LIN {X 0,Y 524.002,Z 585.207,A -85,B 0,C 180,E1 -4848.394,E2 -4848.394} C_VEL
LIN {X 0,Y 523.999,Z 585.214,A -85,B 0,C 180,E1 -4851.516,E2 -4851.516} C_VEL
LIN {X 0,Y 524.093,Z 585.196,A -85,B 0,C 180,E1 -4854.613,E2 -4854.613} C_VEL
LIN {X 0,Y 524.102,Z 585.2,A -85,B 0,C 180,E1 -4857.694,E2 -4857.694} C_VEL
LIN {X 0,Y 524.116,Z 585.194,A -85,B 0,C 180,E1 -4860.768,E2 -4860.768} C_VEL
LIN {X 0,Y 524.067,Z 585.202,A -85,B 0,C 180,E1 -4863.075,E2 -4863.075} C_VEL
LIN {X 0,Y 524.036,Z 585.205,A -85,B 0,C 180,E1 -4866.159,E2 -4866.159} C_VEL
LIN {X 0,Y 523.994,Z 585.212,A -85,B 0,C 180,E1 -4869.262,E2 -4869.262} C_VEL
LIN {X 0,Y 523.997,Z 585.216,A -85,B 0,C 180,E1 -4871.743,E2 -4871.743} C_VEL
LIN {X 0,Y 523.981,Z 585.211,A -85,B 0,C 180,E1 -4875.052,E2 -4875.052} C_VEL
LIN {X 0,Y 523.953,Z 585.22,A -85,B 0,C 180,E1 -4877.969,E2 -4877.969} C_VEL
LIN {X 0,Y 523.961,Z 585.214,A -85,B 0,C 180,E1 -4880.41,E2 -4880.41} C_VEL
LIN {X 0,Y 523.906,Z 585.219,A -85,B 0,C 180,E1 -4882.893,E2 -4882.893} C_VEL
LIN {X 0,Y 523.944,Z 585.217,A -85,B 0,C 180,E1 -4885.419,E2 -4885.419} C_VEL
LIN {X 0,Y 523.96,Z 585.222,A -85,B 0,C 180,E1 -4887.999,E2 -4887.999} C_VEL
LIN {X 0,Y 523.942,Z 585.215,A -85,B 0,C 180,E1 -4890.857,E2 -4890.857} C_VEL
LIN {X 0,Y 523.951,Z 585.218,A -85,B 0,C 180,E1 -4893.735,E2 -4893.735} C_VEL
LIN {X 0,Y 523.915,Z 585.223,A -85,B 0,C 180,E1 -4896.405,E2 -4896.405} C_VEL
LIN {X 0,Y 523.951,Z 585.213,A -85,B 0,C 180,E1 -4899.081,E2 -4899.081} C_VEL
LIN {X 0,Y 523.958,Z 585.221,A -85,B 0,C 180,E1 -4902.118,E2 -4902.118} C_VEL
LIN {X 0,Y 523.947,Z 585.214,A -85,B 0,C 180,E1 -4905.309,E2 -4905.309} C_VEL
LIN {X 0,Y 523.914,Z 585.219,A -85,B 0,C 180,E1 -4906.923,E2 -4906.923} C_VEL
LIN {X 0,Y 523.247,Z 585.302,A -85,B 0,C 180,E1 -4907.565,E2 -4907.565} C_VEL
LIN {X 0,Y 520.402,Z 585.664,A -85,B 0,C 180,E1 -4908.607,E2 -4908.607} C_VEL
LIN {X 0,Y 517.996,Z 585.969,A -85,B 0,C 180,E1 -4909.446,E2 -4909.446} C_VEL
LIN {X 0,Y 516.96,Z 586.095,A -85,B 0,C 180,E1 -4910.093,E2 -4910.093} C_VEL
LIN {X 0,Y 516.874,Z 586.103,A -85,B 0,C 180,E1 -4910.313,E2 -4910.313} C_VEL
LIN {X 0,Y 516.878,Z 586.095,A -85,B 0,C 180,E1 -4913.342,E2 -4913.342} C_VEL
LIN {X 0,Y 516.908,Z 586.095,A -85,B 0,C 180,E1 -4916.122,E2 -4916.122} C_VEL
LIN {X 0,Y 516.887,Z 586.097,A -85,B 0,C 180,E1 -4918.936,E2 -4918.936} C_VEL
LIN {X 0,Y 516.914,Z 586.09,A -85,B 0,C 180,E1 -4921.585,E2 -4921.585} C_VEL
LIN {X 0,Y 516.927,Z 586.092,A -85,B 0,C 180,E1 -4924.211,E2 -4924.211} C_VEL
LIN {X 0,Y 516.868,Z 586.104,A -85,B 0,C 180,E1 -4926.777,E2 -4926.777} C_VEL
LIN {X 0,Y 516.935,Z 586.087,A -85,B 0,C 180,E1 -4929.732,E2 -4929.732} C_VEL
LIN {X 0,Y 516.928,Z 586.095,A -85,B 0,C 180,E1 -4932.597,E2 -4932.597} C_VEL
LIN {X 0,Y 516.939,Z 586.093,A -85,B 0,C 180,E1 -4935.03,E2 -4935.03} C_VEL
LIN {X 0,Y 516.962,Z 586.085,A -85,B 0,C 180,E1 -4938.234,E2 -4938.234} C_VEL
LIN {X 0,Y 516.967,Z 586.086,A -85,B 0,C 180,E1 -4941.4,E2 -4941.4} C_VEL
LIN {X 0,Y 516.999,Z 586.08,A -85,B 0,C 180,E1 -4943.757,E2 -4943.757} C_VEL
LIN {X 0,Y 517.011,Z 586.085,A -85,B 0,C 180,E1 -4946.883,E2 -4946.883} C_VEL
LIN {X 0,Y 517.083,Z 586.069,A -85,B 0,C 180,E1 -4950,E2 -4950} C_VEL
LIN {X 0,Y 517.012,Z 586.088,A -85,B 0,C 180,E1 -4953.117,E2 -4953.117} C_VEL
LIN {X 0,Y 517,Z 586.079,A -85,B 0,C 180,E1 -4956.243,E2 -4956.243} C_VEL
LIN {X 0,Y 516.95,Z 586.093,A -85,B 0,C 180,E1 -4959.389,E2 -4959.389} C_VEL
LIN {X 0,Y 516.949,Z 586.088,A -85,B 0,C 180,E1 -4961.807,E2 -4961.807} C_VEL
LIN {X 0,Y 516.941,Z 586.093,A -85,B 0,C 180,E1 -4965.146,E2 -4965.146} C_VEL
LIN {X 0,Y 516.922,Z 586.089,A -85,B 0,C 180,E1 -4968.222,E2 -4968.222} C_VEL
LIN {X 0,Y 516.908,Z 586.093,A -85,B 0,C 180,E1 -4970.701,E2 -4970.701} C_VEL
LIN {X 0,Y 516.867,Z 586.103,A -85,B 0,C 180,E1 -4973.223,E2 -4973.223} C_VEL
LIN {X 0,Y 516.991,Z 586.242,A -85,B 0,C 180,E1 -4975.877,E2 -4975.877} C_VEL
LIN {X 0,Y 517.471,Z 590.741,A -85,B 0,C 180,E1 -4976.845,E2 -4976.845} C_VEL
LIN {X 0,Y 517.158,Z 604.413,A -85,B 0,C 180,E1 -4979.701,E2 -4979.701} C_VEL
LIN {X 0,Y 519.054,Z 615.156,A -85,B 0,C 180,E1 -4979.913,E2 -4979.913} C_VEL
LIN {X 0,Y 518.599,Z 710.584,A -85,B 0,C 180,E1 -4981.261,E2 -4981.261} C_VEL
LIN {X 0,Y 518.426,Z 723.815,A -85,B 0,C 180,E1 -4981.605,E2 -4981.605} C_VEL
LIN {X 0,Y 518.161,Z 736.677,A -85,B 0,C 180,E1 -4982.107,E2 -4982.107} C_VEL
LIN {X 0,Y 517.866,Z 748.841,A -85,B 0,C 180,E1 -4982.754,E2 -4982.754} C_VEL
LIN {X 0,Y 517.561,Z 759.435,A -85,B 0,C 180,E1 -4983.479,E2 -4983.479} C_VEL
LIN {X 0,Y 517.257,Z 770.01,A -85,B 0,C 180,E1 -4984.382,E2 -4984.382} C_VEL
LIN {X 0,Y 516.977,Z 779.197,A -85,B 0,C 180,E1 -4985.348,E2 -4985.348} C_VEL
LIN {X 0,Y 516.739,Z 787.518,A -85,B 0,C 180,E1 -4986.424,E2 -4986.424} C_VEL
LIN {X 0,Y 516.537,Z 794.357,A -85,B 0,C 180,E1 -4987.507,E2 -4987.507} C_VEL
LIN {X 0,Y 516.404,Z 800.707,A -85,B 0,C 180,E1 -4988.757,E2 -4988.757} C_VEL
LIN {X 0,Y 516.359,Z 804.811,A -85,B 0,C 180,E1 -4989.768,E2 -4989.768} C_VEL
LIN {X 0,Y 516.282,Z 808.167,A -85,B 0,C 180,E1 -4990.798,E2 -4990.798} C_VEL
LIN {X 0,Y 516.285,Z 810.728,A -85,B 0,C 180,E1 -4991.836,E2 -4991.836} C_VEL
LIN {X 0,Y 516.186,Z 812.578,A -85,B 0,C 180,E1 -4992.902,E2 -4992.902} C_VEL
LIN {X 0,Y 516.176,Z 813.697,A -85,B 0,C 180,E1 -4993.977,E2 -4993.977} C_VEL
LIN {X 0,Y 516.182,Z 814.083,A -85,B 0,C 180,E1 -4995.071,E2 -4995.071} C_VEL
LIN {X 0,Y 516.17,Z 813.652,A -85,B 0,C 180,E1 -4996.188,E2 -4996.188} C_VEL
LIN {X 0,Y 516.201,Z 812.387,A -85,B 0,C 180,E1 -4997.323,E2 -4997.323} C_VEL
LIN {X 0,Y 516.292,Z 810.232,A -85,B 0,C 180,E1 -4998.475,E2 -4998.475} C_VEL
LIN {X 0,Y 516.316,Z 807.046,A -85,B 0,C 180,E1 -4999.662,E2 -4999.662} C_VEL
LIN {X 0,Y 516.388,Z 802.692,A -85,B 0,C 180,E1 -5000.873,E2 -5000.873} C_VEL
LIN {X 0,Y 516.52,Z 796.26,A -85,B 0,C 180,E1 -5002.245,E2 -5002.245} C_VEL
LIN {X 0,Y 516.726,Z 789.583,A -85,B 0,C 180,E1 -5003.364,E2 -5003.364} C_VEL
LIN {X 0,Y 516.944,Z 781.446,A -85,B 0,C 180,E1 -5004.472,E2 -5004.472} C_VEL
LIN {X 0,Y 517.213,Z 772.092,A -85,B 0,C 180,E1 -5005.509,E2 -5005.509} C_VEL
LIN {X 0,Y 517.515,Z 762.175,A -85,B 0,C 180,E1 -5006.4,E2 -5006.4} C_VEL
LIN {X 0,Y 517.792,Z 752.322,A -85,B 0,C 180,E1 -5007.118,E2 -5007.118} C_VEL
LIN {X 0,Y 518.056,Z 739.976,A -85,B 0,C 180,E1 -5007.828,E2 -5007.828} C_VEL
LIN {X 0,Y 518.326,Z 727.745,A -85,B 0,C 180,E1 -5008.354,E2 -5008.354} C_VEL
LIN {X 0,Y 518.545,Z 714.491,A -85,B 0,C 180,E1 -5008.744,E2 -5008.744} C_VEL
LIN {X 0,Y 518.678,Z 697.737,A -85,B 0,C 180,E1 -5009.024,E2 -5009.024} C_VEL
LIN {X 0,Y 519.018,Z 614.494,A -85,B 0,C 180,E1 -5010.186,E2 -5010.186} C_VEL
LIN {X 0,Y 517.169,Z 604.571,A -85,B 0,C 180,E1 -5010.395,E2 -5010.395} C_VEL
LIN {X 0,Y 517.523,Z 590.393,A -85,B 0,C 180,E1 -5013.376,E2 -5013.376} C_VEL
LIN {X 0,Y 516.976,Z 586.092,A -85,B 0,C 180,E1 -5014.322,E2 -5014.322} C_VEL
LIN {X 0,Y 516.859,Z 586.1,A -85,B 0,C 180,E1 -5017.622,E2 -5017.622} C_VEL
LIN {X 0,Y 516.922,Z 586.094,A -85,B 0,C 180,E1 -5020.13,E2 -5020.13} C_VEL
LIN {X 0,Y 516.92,Z 586.099,A -85,B 0,C 180,E1 -5022.596,E2 -5022.596} C_VEL
LIN {X 0,Y 516.93,Z 586.094,A -85,B 0,C 180,E1 -5025.03,E2 -5025.03} C_VEL
LIN {X 0,Y 516.993,Z 586.084,A -85,B 0,C 180,E1 -5028.235,E2 -5028.235} C_VEL
LIN {X 0,Y 516.964,Z 586.087,A -85,B 0,C 180,E1 -5031.4,E2 -5031.4} C_VEL
LIN {X 0,Y 517.055,Z 586.08,A -85,B 0,C 180,E1 -5034.541,E2 -5034.541} C_VEL
LIN {X 0,Y 517.075,Z 586.071,A -85,B 0,C 180,E1 -5037.663,E2 -5037.663} C_VEL
LIN {X 0,Y 517.086,Z 586.078,A -85,B 0,C 180,E1 -5040.779,E2 -5040.779} C_VEL
LIN {X 0,Y 517.009,Z 586.084,A -85,B 0,C 180,E1 -5043.117,E2 -5043.117} C_VEL
LIN {X 0,Y 517.006,Z 586.08,A -85,B 0,C 180,E1 -5046.244,E2 -5046.244} C_VEL
LIN {X 0,Y 516.951,Z 586.089,A -85,B 0,C 180,E1 -5049.39,E2 -5049.39} C_VEL
LIN {X 0,Y 516.974,Z 586.084,A -85,B 0,C 180,E1 -5051.825,E2 -5051.825} C_VEL
LIN {X 0,Y 516.934,Z 586.095,A -85,B 0,C 180,E1 -5055.147,E2 -5055.147} C_VEL
LIN {X 0,Y 516.917,Z 586.091,A -85,B 0,C 180,E1 -5058.223,E2 -5058.223} C_VEL
LIN {X 0,Y 516.905,Z 586.095,A -85,B 0,C 180,E1 -5060.702,E2 -5060.702} C_VEL
LIN {X 0,Y 516.903,Z 586.092,A -85,B 0,C 180,E1 -5064.073,E2 -5064.073} C_VEL
LIN {X 0,Y 516.922,Z 586.09,A -85,B 0,C 180,E1 -5066.658,E2 -5066.658} C_VEL
LIN {X 0,Y 516.918,Z 586.095,A -85,B 0,C 180,E1 -5069.527,E2 -5069.527} C_VEL
LIN {X 0,Y 516.895,Z 586.091,A -85,B 0,C 180,E1 -5072.545,E2 -5072.545} C_VEL
LIN {X 0,Y 516.878,Z 586.102,A -85,B 0,C 180,E1 -5075.333,E2 -5075.333} C_VEL
LIN {X 0,Y 516.88,Z 586.096,A -85,B 0,C 180,E1 -5077.945,E2 -5077.945} C_VEL
LIN {X 0,Y 516.881,Z 586.095,A -85,B 0,C 180,E1 -5080.742,E2 -5080.742} C_VEL
LIN {X 0,Y 516.901,Z 586.094,A -85,B 0,C 180,E1 -5082.83,E2 -5082.83} C_VEL
LIN {X 0,Y 516.919,Z 586.094,A -85,B 0,C 180,E1 -5085.011,E2 -5085.011} C_VEL
LIN {X 0,Y 516.919,Z 586.091,A -85,B 0,C 180,E1 -5088.399,E2 -5088.399} C_VEL
LIN {X 0,Y 516.884,Z 586.101,A -85,B 0,C 180,E1 -5091.286,E2 -5091.286} C_VEL
LIN {X 0,Y 516.891,Z 586.096,A -85,B 0,C 180,E1 -5094.222,E2 -5094.222} C_VEL
LIN {X 0,Y 516.896,Z 586.097,A -85,B 0,C 180,E1 -5097.054,E2 -5097.054} C_VEL
LIN {X 0,Y 516.892,Z 586.101,A -85,B 0,C 180,E1 -5099.797,E2 -5099.797} C_VEL
LIN {X 0,Y 516.926,Z 586.093,A -85,B 0,C 180,E1 -5102.468,E2 -5102.468} C_VEL
LIN {X 0,Y 516.978,Z 586.172,A -85,B 0,C 180,E1 -5104.7,E2 -5104.7} C_VEL
LIN {X 0,Y 518.662,Z 595.377,A -85,B 0,C 180,E1 -5106.227,E2 -5106.227} C_VEL
LIN {X 0,Y 518.399,Z 608.933,A -85,B 0,C 180,E1 -5108.32,E2 -5108.32} C_VEL
LIN {X 0,Y 517.851,Z 630.646,A -85,B 0,C 180,E1 -5111.607,E2 -5111.607} C_VEL
LIN {X 0,Y 517.378,Z 650.872,A -85,B 0,C 180,E1 -5114.637,E2 -5114.637} C_VEL
LIN {X 0,Y 519.074,Z 662.348,A -85,B 0,C 180,E1 -5114.85,E2 -5114.85} C_VEL
LIN {X 0,Y 518.618,Z 760.232,A -85,B 0,C 180,E1 -5116.232,E2 -5116.232} C_VEL
LIN {X 0,Y 518.373,Z 773.275,A -85,B 0,C 180,E1 -5116.575,E2 -5116.575} C_VEL
LIN {X 0,Y 518.109,Z 785.905,A -85,B 0,C 180,E1 -5117.067,E2 -5117.067} C_VEL
LIN {X 0,Y 517.868,Z 798.122,A -85,B 0,C 180,E1 -5117.72,E2 -5117.72} C_VEL
LIN {X 0,Y 517.519,Z 810.11,A -85,B 0,C 180,E1 -5118.545,E2 -5118.545} C_VEL
LIN {X 0,Y 517.193,Z 820.364,A -85,B 0,C 180,E1 -5119.43,E2 -5119.43} C_VEL
LIN {X 0,Y 516.939,Z 829.589,A -85,B 0,C 180,E1 -5120.413,E2 -5120.413} C_VEL
LIN {X 0,Y 516.717,Z 838.577,A -85,B 0,C 180,E1 -5121.593,E2 -5121.593} C_VEL
LIN {X 0,Y 516.511,Z 845.809,A -85,B 0,C 180,E1 -5122.77,E2 -5122.77} C_VEL
LIN {X 0,Y 516.427,Z 850.677,A -85,B 0,C 180,E1 -5123.75,E2 -5123.75} C_VEL
LIN {X 0,Y 516.314,Z 855.373,A -85,B 0,C 180,E1 -5124.924,E2 -5124.924} C_VEL
LIN {X 0,Y 516.355,Z 858.958,A -85,B 0,C 180,E1 -5126.098,E2 -5126.098} C_VEL
LIN {X 0,Y 516.283,Z 860.807,A -85,B 0,C 180,E1 -5126.879,E2 -5126.879} C_VEL
LIN {X 0,Y 516.26,Z 862.193,A -85,B 0,C 180,E1 -5127.659,E2 -5127.659} C_VEL
LIN {X 0,Y 516.16,Z 863.785,A -85,B 0,C 180,E1 -5129.22,E2 -5129.22} C_VEL
LIN {X 0,Y 516.154,Z 864,A -85,B 0,C 180,E1 -5130,E2 -5130} C_VEL
LIN {X 0,Y 516.192,Z 863.183,A -85,B 0,C 180,E1 -5131.56,E2 -5131.56} C_VEL
LIN {X 0,Y 516.26,Z 862.195,A -85,B 0,C 180,E1 -5132.341,E2 -5132.341} C_VEL
LIN {X 0,Y 516.283,Z 860.81,A -85,B 0,C 180,E1 -5133.121,E2 -5133.121} C_VEL
LIN {X 0,Y 516.344,Z 857.895,A -85,B 0,C 180,E1 -5134.293,E2 -5134.293} C_VEL
LIN {X 0,Y 516.405,Z 853.948,A -85,B 0,C 180,E1 -5135.467,E2 -5135.467} C_VEL
LIN {X 0,Y 516.486,Z 848.017,A -85,B 0,C 180,E1 -5136.807,E2 -5136.807} C_VEL
LIN {X 0,Y 516.641,Z 841.154,A -85,B 0,C 180,E1 -5138.015,E2 -5138.015} C_VEL
LIN {X 0,Y 516.845,Z 832.837,A -85,B 0,C 180,E1 -5139.194,E2 -5139.194} C_VEL
LIN {X 0,Y 517.076,Z 824.312,A -85,B 0,C 180,E1 -5140.177,E2 -5140.177} C_VEL
LIN {X 0,Y 517.433,Z 813.782,A -85,B 0,C 180,E1 -5141.16,E2 -5141.16} C_VEL
LIN {X 0,Y 517.703,Z 802.188,A -85,B 0,C 180,E1 -5142.029,E2 -5142.029} C_VEL
LIN {X 0,Y 518.026,Z 791.939,A -85,B 0,C 180,E1 -5142.636,E2 -5142.636} C_VEL
LIN {X 0,Y 518.279,Z 780.195,A -85,B 0,C 180,E1 -5143.178,E2 -5143.178} C_VEL
LIN {X 0,Y 518.473,Z 767.577,A -85,B 0,C 180,E1 -5143.597,E2 -5143.597} C_VEL
LIN {X 0,Y 518.677,Z 754.739,A -85,B 0,C 180,E1 -5143.866,E2 -5143.866} C_VEL
LIN {X 0,Y 519.021,Z 661.489,A -85,B 0,C 180,E1 -5145.165,E2 -5145.165} C_VEL
LIN {X 0,Y 517.369,Z 650.938,A -85,B 0,C 180,E1 -5145.374,E2 -5145.374} C_VEL
LIN {X 0,Y 517.925,Z 629.521,A -85,B 0,C 180,E1 -5148.595,E2 -5148.595} C_VEL
LIN {X 0,Y 518.425,Z 609.247,A -85,B 0,C 180,E1 -5151.679,E2 -5151.679} C_VEL
LIN {X 0,Y 518.736,Z 595.718,A -85,B 0,C 180,E1 -5153.769,E2 -5153.769} C_VEL
LIN {X 0,Y 516.951,Z 586.092,A -85,B 0,C 180,E1 -5155.409,E2 -5155.409} C_VEL
LIN {X 0,Y 516.92,Z 586.099,A -85,B 0,C 180,E1 -5158.414,E2 -5158.414} C_VEL
LIN {X 0,Y 516.889,Z 586.096,A -85,B 0,C 180,E1 -5161.109,E2 -5161.109} C_VEL
LIN {X 0,Y 516.912,Z 586.093,A -85,B 0,C 180,E1 -5163.966,E2 -5163.966} C_VEL
LIN {X 0,Y 516.882,Z 586.1,A -85,B 0,C 180,E1 -5166.745,E2 -5166.745} C_VEL
LIN {X 0,Y 516.901,Z 586.092,A -85,B 0,C 180,E1 -5169.718,E2 -5169.718} C_VEL
LIN {X 0,Y 516.915,Z 586.09,A -85,B 0,C 180,E1 -5171.774,E2 -5171.774} C_VEL
LIN {X 0,Y 516.919,Z 586.094,A -85,B 0,C 180,E1 -5175.009,E2 -5175.009} C_VEL
LIN {X 0,Y 516.913,Z 586.095,A -85,B 0,C 180,E1 -5178.397,E2 -5178.397} C_VEL
LIN {X 0,Y 516.879,Z 586.097,A -85,B 0,C 180,E1 -5181.283,E2 -5181.283} C_VEL
LIN {X 0,Y 516.885,Z 586.095,A -85,B 0,C 180,E1 -5184.22,E2 -5184.22} C_VEL
LIN {X 0,Y 516.891,Z 586.099,A -85,B 0,C 180,E1 -5187.052,E2 -5187.052} C_VEL
LIN {X 0,Y 516.895,Z 586.093,A -85,B 0,C 180,E1 -5189.796,E2 -5189.796} C_VEL
LIN {X 0,Y 516.923,Z 586.092,A -85,B 0,C 180,E1 -5192.467,E2 -5192.467} C_VEL
LIN {X 0,Y 516.904,Z 586.1,A -85,B 0,C 180,E1 -5195.071,E2 -5195.071} C_VEL
LIN {X 0,Y 516.878,Z 586.096,A -85,B 0,C 180,E1 -5198.462,E2 -5198.462} C_VEL
LIN {X 0,Y 516.897,Z 586.099,A -85,B 0,C 180,E1 -5200.954,E2 -5200.954} C_VEL
LIN {X 0,Y 516.908,Z 586.096,A -85,B 0,C 180,E1 -5203.41,E2 -5203.41} C_VEL
LIN {X 0,Y 516.886,Z 586.095,A -85,B 0,C 180,E1 -5205.833,E2 -5205.833} C_VEL
LIN {X 0,Y 516.948,Z 586.092,A -85,B 0,C 180,E1 -5209.027,E2 -5209.027} C_VEL
LIN {X 0,Y 516.969,Z 586.083,A -85,B 0,C 180,E1 -5212.186,E2 -5212.186} C_VEL
LIN {X 0,Y 517.038,Z 586.075,A -85,B 0,C 180,E1 -5214.54,E2 -5214.54} C_VEL
LIN {X 0,Y 517.074,Z 586.076,A -85,B 0,C 180,E1 -5217.663,E2 -5217.663} C_VEL
LIN {X 0,Y 517.086,Z 586.07,A -85,B 0,C 180,E1 -5220.778,E2 -5220.778} C_VEL
LIN {X 0,Y 517.008,Z 586.082,A -85,B 0,C 180,E1 -5223.117,E2 -5223.117} C_VEL
LIN {X 0,Y 517,Z 586.08,A -85,B 0,C 180,E1 -5226.243,E2 -5226.243} C_VEL
LIN {X 0,Y 516.948,Z 586.092,A -85,B 0,C 180,E1 -5229.389,E2 -5229.389} C_VEL
LIN {X 0,Y 516.946,Z 586.094,A -85,B 0,C 180,E1 -5231.81,E2 -5231.81} C_VEL
LIN {X 0,Y 516.932,Z 586.09,A -85,B 0,C 180,E1 -5235.146,E2 -5235.146} C_VEL
LIN {X 0,Y 516.915,Z 586.093,A -85,B 0,C 180,E1 -5238.222,E2 -5238.222} C_VEL
LIN {X 0,Y 516.902,Z 586.092,A -85,B 0,C 180,E1 -5240.701,E2 -5240.701} C_VEL
LIN {X 0,Y 516.9,Z 586.099,A -85,B 0,C 180,E1 -5244.072,E2 -5244.072} C_VEL
LIN {X 0,Y 516.919,Z 586.09,A -85,B 0,C 180,E1 -5246.658,E2 -5246.658} C_VEL
LIN {X 0,Y 516.914,Z 586.093,A -85,B 0,C 180,E1 -5249.527,E2 -5249.527} C_VEL
LIN {X 0,Y 516.89,Z 586.096,A -85,B 0,C 180,E1 -5252.545,E2 -5252.545} C_VEL
LIN {X 0,Y 516.873,Z 586.096,A -85,B 0,C 180,E1 -5255.333,E2 -5255.333} C_VEL
LIN {X 0,Y 516.873,Z 586.102,A -85,B 0,C 180,E1 -5257.944,E2 -5257.944} C_VEL
LIN {X 0,Y 516.908,Z 586.093,A -85,B 0,C 180,E1 -5260.739,E2 -5260.739} C_VEL
LIN {X 0,Y 516.875,Z 586.099,A -85,B 0,C 180,E1 -5263.903,E2 -5263.903} C_VEL
LIN {X 0,Y 516.874,Z 586.102,A -85,B 0,C 180,E1 -5266.107,E2 -5266.107} C_VEL
LIN {X 0,Y 516.909,Z 586.099,A -85,B 0,C 180,E1 -5268.399,E2 -5268.399} C_VEL
LIN {X 0,Y 516.874,Z 586.103,A -85,B 0,C 180,E1 -5270.313,E2 -5270.313} C_VEL
LIN {X 0,Y 516.205,Z 586.182,A -85,B 0,C 180,E1 -5270.963,E2 -5270.963} C_VEL
LIN {X 0,Y 513.359,Z 586.537,A -85,B 0,C 180,E1 -5272.019,E2 -5272.019} C_VEL
LIN {X 0,Y 510.952,Z 586.836,A -85,B 0,C 180,E1 -5272.869,E2 -5272.869} C_VEL
LIN {X 0,Y 509.912,Z 586.963,A -85,B 0,C 180,E1 -5273.526,E2 -5273.526} C_VEL
LIN {X 0,Y 509.825,Z 586.974,A -85,B 0,C 180,E1 -5273.748,E2 -5273.748} C_VEL
LIN {X 0,Y 509.858,Z 586.978,A -85,B 0,C 180,E1 -5276.54,E2 -5276.54} C_VEL
LIN {X 0,Y 509.84,Z 586.972,A -85,B 0,C 180,E1 -5279.335,E2 -5279.335} C_VEL
LIN {X 0,Y 509.889,Z 586.968,A -85,B 0,C 180,E1 -5282.055,E2 -5282.055} C_VEL
LIN {X 0,Y 509.872,Z 586.976,A -85,B 0,C 180,E1 -5284.704,E2 -5284.704} C_VEL
LIN {X 0,Y 509.832,Z 586.973,A -85,B 0,C 180,E1 -5287.455,E2 -5287.455} C_VEL
LIN {X 0,Y 509.913,Z 586.962,A -85,B 0,C 180,E1 -5289.845,E2 -5289.845} C_VEL
LIN {X 0,Y 509.883,Z 586.97,A -85,B 0,C 180,E1 -5293.175,E2 -5293.175} C_VEL
LIN {X 0,Y 509.861,Z 586.969,A -85,B 0,C 180,E1 -5295.634,E2 -5295.634} C_VEL
LIN {X 0,Y 509.898,Z 586.965,A -85,B 0,C 180,E1 -5298.123,E2 -5298.123} C_VEL
LIN {X 0,Y 509.914,Z 586.966,A -85,B 0,C 180,E1 -5301.28,E2 -5301.28} C_VEL
LIN {X 0,Y 509.95,Z 586.958,A -85,B 0,C 180,E1 -5303.67,E2 -5303.67} C_VEL
LIN {X 0,Y 509.954,Z 586.964,A -85,B 0,C 180,E1 -5306.84,E2 -5306.84} C_VEL
LIN {X 0,Y 510.062,Z 586.951,A -85,B 0,C 180,E1 -5309.211,E2 -5309.211} C_VEL
LIN {X 0,Y 510.053,Z 586.945,A -85,B 0,C 180,E1 -5312.369,E2 -5312.369} C_VEL
LIN {X 0,Y 509.977,Z 586.958,A -85,B 0,C 180,E1 -5315.536,E2 -5315.536} C_VEL
LIN {X 0,Y 509.949,Z 586.959,A -85,B 0,C 180,E1 -5317.921,E2 -5317.921} C_VEL
LIN {X 0,Y 509.91,Z 586.97,A -85,B 0,C 180,E1 -5321.125,E2 -5321.125} C_VEL
LIN {X 0,Y 509.861,Z 586.969,A -85,B 0,C 180,E1 -5324.366,E2 -5324.366} C_VEL
LIN {X 0,Y 509.899,Z 586.971,A -85,B 0,C 180,E1 -5327.651,E2 -5327.651} C_VEL
LIN {X 0,Y 509.882,Z 586.968,A -85,B 0,C 180,E1 -5330.401,E2 -5330.401} C_VEL
LIN {X 0,Y 509.826,Z 586.983,A -85,B 0,C 180,E1 -5333.563,E2 -5333.563} C_VEL
LIN {X 0,Y 509.935,Z 587.072,A -85,B 0,C 180,E1 -5335.73,E2 -5335.73} C_VEL
LIN {X 0,Y 510.496,Z 591.533,A -85,B 0,C 180,E1 -5336.7,E2 -5336.7} C_VEL
LIN {X 0,Y 510.184,Z 604.679,A -85,B 0,C 180,E1 -5339.474,E2 -5339.474} C_VEL
LIN {X 0,Y 512.213,Z 615.808,A -85,B 0,C 180,E1 -5339.713,E2 -5339.713} C_VEL
LIN {X 0,Y 511.703,Z 711.341,A -85,B 0,C 180,E1 -5341.086,E2 -5341.086} C_VEL
LIN {X 0,Y 511.476,Z 724.784,A -85,B 0,C 180,E1 -5341.446,E2 -5341.446} C_VEL
LIN {X 0,Y 511.258,Z 737.546,A -85,B 0,C 180,E1 -5341.959,E2 -5341.959} C_VEL
LIN {X 0,Y 510.941,Z 749.519,A -85,B 0,C 180,E1 -5342.613,E2 -5342.613} C_VEL
LIN {X 0,Y 510.578,Z 760.801,A -85,B 0,C 180,E1 -5343.407,E2 -5343.407} C_VEL
LIN {X 0,Y 510.27,Z 770.675,A -85,B 0,C 180,E1 -5344.272,E2 -5344.272} C_VEL
LIN {X 0,Y 509.982,Z 779.742,A -85,B 0,C 180,E1 -5345.244,E2 -5345.244} C_VEL
LIN {X 0,Y 509.718,Z 788.197,A -85,B 0,C 180,E1 -5346.361,E2 -5346.361} C_VEL
LIN {X 0,Y 509.477,Z 795.569,A -85,B 0,C 180,E1 -5347.565,E2 -5347.565} C_VEL
LIN {X 0,Y 509.336,Z 802.001,A -85,B 0,C 180,E1 -5348.889,E2 -5348.889} C_VEL
LIN {X 0,Y 509.249,Z 807.596,A -85,B 0,C 180,E1 -5350.437,E2 -5350.437} C_VEL
LIN {X 0,Y 509.199,Z 811.115,A -85,B 0,C 180,E1 -5351.815,E2 -5351.815} C_VEL
LIN {X 0,Y 509.117,Z 813.064,A -85,B 0,C 180,E1 -5352.978,E2 -5352.978} C_VEL
LIN {X 0,Y 509.089,Z 814.135,A -85,B 0,C 180,E1 -5354.122,E2 -5354.122} C_VEL
LIN {X 0,Y 509.092,Z 814.393,A -85,B 0,C 180,E1 -5355.248,E2 -5355.248} C_VEL
LIN {X 0,Y 509.101,Z 813.892,A -85,B 0,C 180,E1 -5356.352,E2 -5356.352} C_VEL
LIN {X 0,Y 509.119,Z 812.617,A -85,B 0,C 180,E1 -5357.437,E2 -5357.437} C_VEL
LIN {X 0,Y 509.206,Z 810.604,A -85,B 0,C 180,E1 -5358.511,E2 -5358.511} C_VEL
LIN {X 0,Y 509.249,Z 807.894,A -85,B 0,C 180,E1 -5359.562,E2 -5359.562} C_VEL
LIN {X 0,Y 509.309,Z 803.431,A -85,B 0,C 180,E1 -5360.854,E2 -5360.854} C_VEL
LIN {X 0,Y 509.475,Z 797.14,A -85,B 0,C 180,E1 -5362.239,E2 -5362.239} C_VEL
LIN {X 0,Y 509.692,Z 790.553,A -85,B 0,C 180,E1 -5363.382,E2 -5363.382} C_VEL
LIN {X 0,Y 509.929,Z 781.546,A -85,B 0,C 180,E1 -5364.63,E2 -5364.63} C_VEL
LIN {X 0,Y 510.275,Z 771.685,A -85,B 0,C 180,E1 -5365.726,E2 -5365.726} C_VEL
LIN {X 0,Y 510.546,Z 762.048,A -85,B 0,C 180,E1 -5366.591,E2 -5366.591} C_VEL
LIN {X 0,Y 510.873,Z 751.097,A -85,B 0,C 180,E1 -5367.381,E2 -5367.381} C_VEL
LIN {X 0,Y 511.178,Z 739.498,A -85,B 0,C 180,E1 -5368.04,E2 -5368.04} C_VEL
LIN {X 0,Y 511.452,Z 726.716,A -85,B 0,C 180,E1 -5368.58,E2 -5368.58} C_VEL
LIN {X 0,Y 511.655,Z 713.696,A -85,B 0,C 180,E1 -5368.954,E2 -5368.954} C_VEL
LIN {X 0,Y 511.857,Z 692.969,A -85,B 0,C 180,E1 -5369.282,E2 -5369.282} C_VEL
LIN {X 0,Y 512.206,Z 615.416,A -85,B 0,C 180,E1 -5370.383,E2 -5370.383} C_VEL
LIN {X 0,Y 510.191,Z 604.951,A -85,B 0,C 180,E1 -5370.611,E2 -5370.611} C_VEL
LIN {X 0,Y 510.541,Z 591.452,A -85,B 0,C 180,E1 -5373.477,E2 -5373.477} C_VEL
LIN {X 0,Y 509.922,Z 586.971,A -85,B 0,C 180,E1 -5374.488,E2 -5374.488} C_VEL
LIN {X 0,Y 509.825,Z 586.977,A -85,B 0,C 180,E1 -5377.455,E2 -5377.455} C_VEL
LIN {X 0,Y 509.906,Z 586.966,A -85,B 0,C 180,E1 -5379.845,E2 -5379.845} C_VEL
LIN {X 0,Y 509.876,Z 586.971,A -85,B 0,C 180,E1 -5383.175,E2 -5383.175} C_VEL
LIN {X 0,Y 509.854,Z 586.972,A -85,B 0,C 180,E1 -5385.634,E2 -5385.634} C_VEL
LIN {X 0,Y 509.916,Z 586.971,A -85,B 0,C 180,E1 -5388.875,E2 -5388.875} C_VEL
LIN {X 0,Y 509.942,Z 586.962,A -85,B 0,C 180,E1 -5392.079,E2 -5392.079} C_VEL
LIN {X 0,Y 510.001,Z 586.957,A -85,B 0,C 180,E1 -5394.465,E2 -5394.465} C_VEL
LIN {X 0,Y 510.048,Z 586.947,A -85,B 0,C 180,E1 -5397.631,E2 -5397.631} C_VEL
LIN {X 0,Y 510.056,Z 586.953,A -85,B 0,C 180,E1 -5400.79,E2 -5400.79} C_VEL
LIN {X 0,Y 509.952,Z 586.962,A -85,B 0,C 180,E1 -5403.161,E2 -5403.161} C_VEL
LIN {X 0,Y 509.973,Z 586.957,A -85,B 0,C 180,E1 -5406.33,E2 -5406.33} C_VEL
LIN {X 0,Y 509.911,Z 586.969,A -85,B 0,C 180,E1 -5408.721,E2 -5408.721} C_VEL
LIN {X 0,Y 509.942,Z 586.959,A -85,B 0,C 180,E1 -5411.931,E2 -5411.931} C_VEL
LIN {X 0,Y 509.884,Z 586.971,A -85,B 0,C 180,E1 -5415.242,E2 -5415.242} C_VEL
LIN {X 0,Y 509.88,Z 586.967,A -85,B 0,C 180,E1 -5418.002,E2 -5418.002} C_VEL
LIN {X 0,Y 509.842,Z 586.979,A -85,B 0,C 180,E1 -5421.002,E2 -5421.002} C_VEL
LIN {X 0,Y 509.862,Z 586.97,A -85,B 0,C 180,E1 -5424.427,E2 -5424.427} C_VEL
LIN {X 0,Y 509.881,Z 586.972,A -85,B 0,C 180,E1 -5427.056,E2 -5427.056} C_VEL
LIN {X 0,Y 509.874,Z 586.969,A -85,B 0,C 180,E1 -5429.75,E2 -5429.75} C_VEL
LIN {X 0,Y 509.871,Z 586.968,A -85,B 0,C 180,E1 -5432.776,E2 -5432.776} C_VEL
LIN {X 0,Y 509.837,Z 586.978,A -85,B 0,C 180,E1 -5435.582,E2 -5435.582} C_VEL
LIN {X 0,Y 509.848,Z 586.97,A -85,B 0,C 180,E1 -5438.339,E2 -5438.339} C_VEL
LIN {X 0,Y 509.854,Z 586.978,A -85,B 0,C 180,E1 -5441.426,E2 -5441.426} C_VEL
LIN {X 0,Y 509.853,Z 586.972,A -85,B 0,C 180,E1 -5444.669,E2 -5444.669} C_VEL
LIN {X 0,Y 509.858,Z 586.972,A -85,B 0,C 180,E1 -5448.104,E2 -5448.104} C_VEL
LIN {X 0,Y 509.858,Z 586.971,A -85,B 0,C 180,E1 -5450.65,E2 -5450.65} C_VEL
LIN {X 0,Y 509.835,Z 586.982,A -85,B 0,C 180,E1 -5453.649,E2 -5453.649} C_VEL
LIN {X 0,Y 509.861,Z 586.972,A -85,B 0,C 180,E1 -5456.54,E2 -5456.54} C_VEL
LIN {X 0,Y 509.845,Z 586.976,A -85,B 0,C 180,E1 -5459.335,E2 -5459.335} C_VEL
LIN {X 0,Y 509.893,Z 586.973,A -85,B 0,C 180,E1 -5462.055,E2 -5462.055} C_VEL
LIN {X 0,Y 509.922,Z 587.026,A -85,B 0,C 180,E1 -5464.516,E2 -5464.516} C_VEL
LIN {X 0,Y 511.688,Z 596.418,A -85,B 0,C 180,E1 -5466.098,E2 -5466.098} C_VEL
LIN {X 0,Y 511.516,Z 607.216,A -85,B 0,C 180,E1 -5467.801,E2 -5467.801} C_VEL
LIN {X 0,Y 510.905,Z 628.925,A -85,B 0,C 180,E1 -5471.14,E2 -5471.14} C_VEL
LIN {X 0,Y 510.369,Z 650.05,A -85,B 0,C 180,E1 -5474.356,E2 -5474.356} C_VEL
LIN {X 0,Y 510.383,Z 650.663,A -85,B 0,C 180,E1 -5474.424,E2 -5474.424} C_VEL
LIN {X 0,Y 512.186,Z 663.119,A -85,B 0,C 180,E1 -5474.66,E2 -5474.66} C_VEL
LIN {X 0,Y 511.723,Z 759.602,A -85,B 0,C 180,E1 -5476.043,E2 -5476.043} C_VEL
LIN {X 0,Y 511.459,Z 772.727,A -85,B 0,C 180,E1 -5476.39,E2 -5476.39} C_VEL
LIN {X 0,Y 511.164,Z 785.403,A -85,B 0,C 180,E1 -5476.888,E2 -5476.888} C_VEL
LIN {X 0,Y 510.896,Z 797.381,A -85,B 0,C 180,E1 -5477.532,E2 -5477.532} C_VEL
LIN {X 0,Y 510.529,Z 809.668,A -85,B 0,C 180,E1 -5478.386,E2 -5478.386} C_VEL
LIN {X 0,Y 510.175,Z 819.944,A -85,B 0,C 180,E1 -5479.282,E2 -5479.282} C_VEL
LIN {X 0,Y 509.912,Z 829.184,A -85,B 0,C 180,E1 -5480.28,E2 -5480.28} C_VEL
LIN {X 0,Y 509.657,Z 838.183,A -85,B 0,C 180,E1 -5481.475,E2 -5481.475} C_VEL
LIN {X 0,Y 509.438,Z 845.428,A -85,B 0,C 180,E1 -5482.669,E2 -5482.669} C_VEL
LIN {X 0,Y 509.327,Z 850.315,A -85,B 0,C 180,E1 -5483.662,E2 -5483.662} C_VEL
LIN {X 0,Y 509.248,Z 855.067,A -85,B 0,C 180,E1 -5484.854,E2 -5484.854} C_VEL
LIN {X 0,Y 509.253,Z 858.701,A -85,B 0,C 180,E1 -5486.043,E2 -5486.043} C_VEL
LIN {X 0,Y 509.201,Z 860.573,A -85,B 0,C 180,E1 -5486.835,E2 -5486.835} C_VEL
LIN {X 0,Y 509.189,Z 861.977,A -85,B 0,C 180,E1 -5487.627,E2 -5487.627} C_VEL
LIN {X 0,Y 509.073,Z 863.585,A -85,B 0,C 180,E1 -5489.209,E2 -5489.209} C_VEL
LIN {X 0,Y 509.065,Z 863.803,A -85,B 0,C 180,E1 -5490,E2 -5490} C_VEL
LIN {X 0,Y 509.112,Z 862.979,A -85,B 0,C 180,E1 -5491.582,E2 -5491.582} C_VEL
LIN {X 0,Y 509.189,Z 861.984,A -85,B 0,C 180,E1 -5492.373,E2 -5492.373} C_VEL
LIN {X 0,Y 509.201,Z 860.582,A -85,B 0,C 180,E1 -5493.165,E2 -5493.165} C_VEL
LIN {X 0,Y 509.23,Z 857.633,A -85,B 0,C 180,E1 -5494.353,E2 -5494.353} C_VEL
LIN {X 0,Y 509.322,Z 853.643,A -85,B 0,C 180,E1 -5495.543,E2 -5495.543} C_VEL
LIN {X 0,Y 509.405,Z 847.958,A -85,B 0,C 180,E1 -5496.844,E2 -5496.844} C_VEL
LIN {X 0,Y 509.585,Z 840.793,A -85,B 0,C 180,E1 -5498.127,E2 -5498.127} C_VEL
LIN {X 0,Y 509.794,Z 832.468,A -85,B 0,C 180,E1 -5499.322,E2 -5499.322} C_VEL
LIN {X 0,Y 510.039,Z 823.931,A -85,B 0,C 180,E1 -5500.319,E2 -5500.319} C_VEL
LIN {X 0,Y 510.434,Z 813.39,A -85,B 0,C 180,E1 -5501.315,E2 -5501.315} C_VEL
LIN {X 0,Y 510.714,Z 801.782,A -85,B 0,C 180,E1 -5502.196,E2 -5502.196} C_VEL
LIN {X 0,Y 511.058,Z 791.514,A -85,B 0,C 180,E1 -5502.811,E2 -5502.811} C_VEL
LIN {X 0,Y 511.357,Z 779.731,A -85,B 0,C 180,E1 -5503.36,E2 -5503.36} C_VEL
LIN {X 0,Y 511.588,Z 767.063,A -85,B 0,C 180,E1 -5503.784,E2 -5503.784} C_VEL
LIN {X 0,Y 511.798,Z 754.125,A -85,B 0,C 180,E1 -5504.056,E2 -5504.056} C_VEL
LIN {X 0,Y 512.064,Z 661.665,A -85,B 0,C 180,E1 -5505.367,E2 -5505.367} C_VEL
LIN {X 0,Y 510.37,Z 650.605,A -85,B 0,C 180,E1 -5505.592,E2 -5505.592} C_VEL
LIN {X 0,Y 510.952,Z 629.255,A -85,B 0,C 180,E1 -5508.858,E2 -5508.858} C_VEL
LIN {X 0,Y 511.475,Z 610.331,A -85,B 0,C 180,E1 -5511.777,E2 -5511.777} C_VEL
LIN {X 0,Y 511.78,Z 596.828,A -85,B 0,C 180,E1 -5513.897,E2 -5513.897} C_VEL
LIN {X 0,Y 509.916,Z 586.97,A -85,B 0,C 180,E1 -5515.594,E2 -5515.594} C_VEL
LIN {X 0,Y 509.877,Z 586.972,A -85,B 0,C 180,E1 -5518.843,E2 -5518.843} C_VEL
LIN {X 0,Y 509.821,Z 586.976,A -85,B 0,C 180,E1 -5521.589,E2 -5521.589} C_VEL
LIN {X 0,Y 509.853,Z 586.979,A -85,B 0,C 180,E1 -5524.412,E2 -5524.412} C_VEL
LIN {X 0,Y 509.818,Z 586.974,A -85,B 0,C 180,E1 -5527.34,E2 -5527.34} C_VEL
LIN {X 0,Y 509.859,Z 586.976,A -85,B 0,C 180,E1 -5530.379,E2 -5530.379} C_VEL
LIN {X 0,Y 509.821,Z 586.977,A -85,B 0,C 180,E1 -5533.061,E2 -5533.061} C_VEL
LIN {X 0,Y 509.827,Z 586.973,A -85,B 0,C 180,E1 -5535.791,E2 -5535.791} C_VEL
LIN {X 0,Y 509.854,Z 586.977,A -85,B 0,C 180,E1 -5538.574,E2 -5538.574} C_VEL
LIN {X 0,Y 509.848,Z 586.97,A -85,B 0,C 180,E1 -5541.785,E2 -5541.785} C_VEL
LIN {X 0,Y 509.84,Z 586.978,A -85,B 0,C 180,E1 -5544.622,E2 -5544.622} C_VEL
LIN {X 0,Y 509.859,Z 586.97,A -85,B 0,C 180,E1 -5547.48,E2 -5547.48} C_VEL
LIN {X 0,Y 509.875,Z 586.968,A -85,B 0,C 180,E1 -5550.268,E2 -5550.268} C_VEL
LIN {X 0,Y 509.88,Z 586.976,A -85,B 0,C 180,E1 -5552.944,E2 -5552.944} C_VEL
LIN {X 0,Y 509.862,Z 586.971,A -85,B 0,C 180,E1 -5555.573,E2 -5555.573} C_VEL
LIN {X 0,Y 509.842,Z 586.98,A -85,B 0,C 180,E1 -5558.998,E2 -5558.998} C_VEL
LIN {X 0,Y 509.88,Z 586.967,A -85,B 0,C 180,E1 -5561.998,E2 -5561.998} C_VEL
LIN {X 0,Y 509.901,Z 586.968,A -85,B 0,C 180,E1 -5564.818,E2 -5564.818} C_VEL
LIN {X 0,Y 509.896,Z 586.965,A -85,B 0,C 180,E1 -5568.121,E2 -5568.121} C_VEL
LIN {X 0,Y 509.909,Z 586.972,A -85,B 0,C 180,E1 -5571.279,E2 -5571.279} C_VEL
LIN {X 0,Y 509.972,Z 586.959,A -85,B 0,C 180,E1 -5573.67,E2 -5573.67} C_VEL
LIN {X 0,Y 510.045,Z 586.952,A -85,B 0,C 180,E1 -5577.63,E2 -5577.63} C_VEL
LIN {X 0,Y 510.056,Z 586.945,A -85,B 0,C 180,E1 -5580.789,E2 -5580.789} C_VEL
LIN {X 0,Y 509.95,Z 586.962,A -85,B 0,C 180,E1 -5583.16,E2 -5583.16} C_VEL
LIN {X 0,Y 509.968,Z 586.956,A -85,B 0,C 180,E1 -5586.329,E2 -5586.329} C_VEL
LIN {X 0,Y 509.909,Z 586.963,A -85,B 0,C 180,E1 -5588.72,E2 -5588.72} C_VEL
LIN {X 0,Y 509.894,Z 586.97,A -85,B 0,C 180,E1 -5591.931,E2 -5591.931} C_VEL
LIN {X 0,Y 509.882,Z 586.969,A -85,B 0,C 180,E1 -5595.242,E2 -5595.242} C_VEL
LIN {X 0,Y 509.877,Z 586.973,A -85,B 0,C 180,E1 -5598.001,E2 -5598.001} C_VEL
LIN {X 0,Y 509.84,Z 586.972,A -85,B 0,C 180,E1 -5601.002,E2 -5601.002} C_VEL
LIN {X 0,Y 509.859,Z 586.971,A -85,B 0,C 180,E1 -5604.426,E2 -5604.426} C_VEL
LIN {X 0,Y 509.877,Z 586.967,A -85,B 0,C 180,E1 -5607.056,E2 -5607.056} C_VEL
LIN {X 0,Y 509.871,Z 586.973,A -85,B 0,C 180,E1 -5609.75,E2 -5609.75} C_VEL
LIN {X 0,Y 509.866,Z 586.969,A -85,B 0,C 180,E1 -5612.775,E2 -5612.775} C_VEL
LIN {X 0,Y 509.833,Z 586.974,A -85,B 0,C 180,E1 -5615.582,E2 -5615.582} C_VEL
LIN {X 0,Y 509.85,Z 586.977,A -85,B 0,C 180,E1 -5618.337,E2 -5618.337} C_VEL
LIN {X 0,Y 509.864,Z 586.969,A -85,B 0,C 180,E1 -5621.424,E2 -5621.424} C_VEL
LIN {X 0,Y 509.848,Z 586.974,A -85,B 0,C 180,E1 -5624.668,E2 -5624.668} C_VEL
LIN {X 0,Y 509.853,Z 586.976,A -85,B 0,C 180,E1 -5628.103,E2 -5628.103} C_VEL
LIN {X 0,Y 509.84,Z 586.977,A -85,B 0,C 180,E1 -5630.648,E2 -5630.648} C_VEL
LIN {X 0,Y 509.825,Z 586.974,A -85,B 0,C 180,E1 -5633.748,E2 -5633.748} C_VEL
LIN {X 0,Y 509.16,Z 587.065,A -85,B 0,C 180,E1 -5634.408,E2 -5634.408} C_VEL
LIN {X 0,Y 506.341,Z 587.414,A -85,B 0,C 180,E1 -5635.48,E2 -5635.48} C_VEL
LIN {X 0,Y 503.948,Z 587.713,A -85,B 0,C 180,E1 -5636.343,E2 -5636.343} C_VEL
LIN {X 0,Y 502.899,Z 587.838,A -85,B 0,C 180,E1 -5637.009,E2 -5637.009} C_VEL
LIN {X 0,Y 502.803,Z 587.849,A -85,B 0,C 180,E1 -5637.235,E2 -5637.235} C_VEL
LIN {X 0,Y 502.809,Z 587.85,A -85,B 0,C 180,E1 -5640.065,E2 -5640.065} C_VEL
LIN {X 0,Y 502.829,Z 587.854,A -85,B 0,C 180,E1 -5642.534,E2 -5642.534} C_VEL
LIN {X 0,Y 502.824,Z 587.846,A -85,B 0,C 180,E1 -5645.299,E2 -5645.299} C_VEL
LIN {X 0,Y 502.78,Z 587.851,A -85,B 0,C 180,E1 -5647.827,E2 -5647.827} C_VEL
LIN {X 0,Y 502.822,Z 587.85,A -85,B 0,C 180,E1 -5650.401,E2 -5650.401} C_VEL
LIN {X 0,Y 502.833,Z 587.851,A -85,B 0,C 180,E1 -5652.932,E2 -5652.932} C_VEL
LIN {X 0,Y 502.842,Z 587.845,A -85,B 0,C 180,E1 -5655.429,E2 -5655.429} C_VEL
LIN {X 0,Y 502.874,Z 587.846,A -85,B 0,C 180,E1 -5658.717,E2 -5658.717} C_VEL
LIN {X 0,Y 502.899,Z 587.836,A -85,B 0,C 180,E1 -5661.967,E2 -5661.967} C_VEL
LIN {X 0,Y 502.931,Z 587.834,A -85,B 0,C 180,E1 -5664.387,E2 -5664.387} C_VEL
LIN {X 0,Y 503.023,Z 587.822,A -85,B 0,C 180,E1 -5667.598,E2 -5667.598} C_VEL
LIN {X 0,Y 503.025,Z 587.82,A -85,B 0,C 180,E1 -5670,E2 -5670} C_VEL
LIN {X 0,Y 503.023,Z 587.821,A -85,B 0,C 180,E1 -5672.402,E2 -5672.402} C_VEL
LIN {X 0,Y 502.931,Z 587.835,A -85,B 0,C 180,E1 -5675.613,E2 -5675.613} C_VEL
LIN {X 0,Y 502.899,Z 587.836,A -85,B 0,C 180,E1 -5678.033,E2 -5678.033} C_VEL
LIN {X 0,Y 502.874,Z 587.849,A -85,B 0,C 180,E1 -5681.283,E2 -5681.283} C_VEL
LIN {X 0,Y 502.842,Z 587.844,A -85,B 0,C 180,E1 -5684.571,E2 -5684.571} C_VEL
LIN {X 0,Y 502.858,Z 587.844,A -85,B 0,C 180,E1 -5687.907,E2 -5687.907} C_VEL
LIN {X 0,Y 502.824,Z 587.848,A -85,B 0,C 180,E1 -5690.536,E2 -5690.536} C_VEL
LIN {X 0,Y 502.79,Z 587.855,A -85,B 0,C 180,E1 -5693.04,E2 -5693.04} C_VEL
LIN {X 0,Y 502.91,Z 587.95,A -85,B 0,C 180,E1 -5695.588,E2 -5695.588} C_VEL
LIN {X 0,Y 503.503,Z 593.056,A -85,B 0,C 180,E1 -5696.707,E2 -5696.707} C_VEL
LIN {X 0,Y 503.222,Z 605.04,A -85,B 0,C 180,E1 -5699.262,E2 -5699.262} C_VEL
LIN {X 0,Y 505.39,Z 616.684,A -85,B 0,C 180,E1 -5699.511,E2 -5699.511} C_VEL
LIN {X 0,Y 504.814,Z 711.512,A -85,B 0,C 180,E1 -5700.893,E2 -5700.893} C_VEL
LIN {X 0,Y 504.584,Z 725.256,A -85,B 0,C 180,E1 -5701.267,E2 -5701.267} C_VEL
LIN {X 0,Y 504.363,Z 738.017,A -85,B 0,C 180,E1 -5701.79,E2 -5701.79} C_VEL
LIN {X 0,Y 504.016,Z 750.198,A -85,B 0,C 180,E1 -5702.468,E2 -5702.468} C_VEL
LIN {X 0,Y 503.606,Z 761.436,A -85,B 0,C 180,E1 -5703.273,E2 -5703.273} C_VEL
LIN {X 0,Y 503.249,Z 772.294,A -85,B 0,C 180,E1 -5704.254,E2 -5704.254} C_VEL
LIN {X 0,Y 502.956,Z 780.761,A -85,B 0,C 180,E1 -5705.197,E2 -5705.197} C_VEL
LIN {X 0,Y 502.662,Z 789.93,A -85,B 0,C 180,E1 -5706.456,E2 -5706.456} C_VEL
LIN {X 0,Y 502.428,Z 796.273,A -85,B 0,C 180,E1 -5707.532,E2 -5707.532} C_VEL
LIN {X 0,Y 502.301,Z 801.844,A -85,B 0,C 180,E1 -5708.693,E2 -5708.693} C_VEL
LIN {X 0,Y 502.207,Z 806.998,A -85,B 0,C 180,E1 -5710.07,E2 -5710.07} C_VEL
LIN {X 0,Y 502.13,Z 811.118,A -85,B 0,C 180,E1 -5711.617,E2 -5711.617} C_VEL
LIN {X 0,Y 502.076,Z 812.277,A -85,B 0,C 180,E1 -5712.212,E2 -5712.212} C_VEL
LIN {X 0,Y 502.026,Z 813.828,A -85,B 0,C 180,E1 -5713.31,E2 -5713.31} C_VEL
LIN {X 0,Y 502.001,Z 814.656,A -85,B 0,C 180,E1 -5714.44,E2 -5714.44} C_VEL
LIN {X 0,Y 502.002,Z 814.675,A -85,B 0,C 180,E1 -5715.574,E2 -5715.574} C_VEL
LIN {X 0,Y 502.026,Z 813.901,A -85,B 0,C 180,E1 -5716.714,E2 -5716.714} C_VEL
LIN {X 0,Y 502.086,Z 812.271,A -85,B 0,C 180,E1 -5717.89,E2 -5717.89} C_VEL
LIN {X 0,Y 502.136,Z 809.687,A -85,B 0,C 180,E1 -5719.093,E2 -5719.093} C_VEL
LIN {X 0,Y 502.207,Z 806.015,A -85,B 0,C 180,E1 -5720.324,E2 -5720.324} C_VEL
LIN {X 0,Y 502.375,Z 800.133,A -85,B 0,C 180,E1 -5721.793,E2 -5721.793} C_VEL
LIN {X 0,Y 502.553,Z 793.684,A -85,B 0,C 180,E1 -5723.035,E2 -5723.035} C_VEL
LIN {X 0,Y 502.77,Z 786.371,A -85,B 0,C 180,E1 -5724.168,E2 -5724.168} C_VEL
LIN {X 0,Y 503.093,Z 777.265,A -85,B 0,C 180,E1 -5725.312,E2 -5725.312} C_VEL
LIN {X 0,Y 503.409,Z 767.919,A -85,B 0,C 180,E1 -5726.268,E2 -5726.268} C_VEL
LIN {X 0,Y 503.792,Z 757.07,A -85,B 0,C 180,E1 -5727.159,E2 -5727.159} C_VEL
LIN {X 0,Y 504.163,Z 744.736,A -85,B 0,C 180,E1 -5727.955,E2 -5727.955} C_VEL
LIN {X 0,Y 504.506,Z 732.141,A -85,B 0,C 180,E1 -5728.566,E2 -5728.566} C_VEL
LIN {X 0,Y 504.668,Z 719.279,A -85,B 0,C 180,E1 -5729.01,E2 -5729.01} C_VEL
LIN {X 0,Y 504.909,Z 705.74,A -85,B 0,C 180,E1 -5729.297,E2 -5729.297} C_VEL
LIN {X 0,Y 505.356,Z 616.319,A -85,B 0,C 180,E1 -5730.588,E2 -5730.588} C_VEL
LIN {X 0,Y 503.252,Z 605.32,A -85,B 0,C 180,E1 -5730.835,E2 -5730.835} C_VEL
LIN {X 0,Y 503.566,Z 593.002,A -85,B 0,C 180,E1 -5733.474,E2 -5733.474} C_VEL
LIN {X 0,Y 502.867,Z 587.85,A -85,B 0,C 180,E1 -5734.659,E2 -5734.659} C_VEL
LIN {X 0,Y 502.774,Z 587.856,A -85,B 0,C 180,E1 -5737.827,E2 -5737.827} C_VEL
LIN {X 0,Y 502.816,Z 587.854,A -85,B 0,C 180,E1 -5740.4,E2 -5740.4} C_VEL
LIN {X 0,Y 502.826,Z 587.852,A -85,B 0,C 180,E1 -5742.932,E2 -5742.932} C_VEL
LIN {X 0,Y 502.834,Z 587.847,A -85,B 0,C 180,E1 -5745.429,E2 -5745.429} C_VEL
LIN {X 0,Y 502.885,Z 587.847,A -85,B 0,C 180,E1 -5748.717,E2 -5748.717} C_VEL
LIN {X 0,Y 502.892,Z 587.839,A -85,B 0,C 180,E1 -5751.967,E2 -5751.967} C_VEL
LIN {X 0,Y 502.953,Z 587.834,A -85,B 0,C 180,E1 -5754.387,E2 -5754.387} C_VEL
LIN {X 0,Y 503.019,Z 587.823,A -85,B 0,C 180,E1 -5757.598,E2 -5757.598} C_VEL
LIN {X 0,Y 503.026,Z 587.829,A -85,B 0,C 180,E1 -5760.801,E2 -5760.801} C_VEL
LIN {X 0,Y 502.895,Z 587.841,A -85,B 0,C 180,E1 -5763.205,E2 -5763.205} C_VEL
LIN {X 0,Y 502.922,Z 587.836,A -85,B 0,C 180,E1 -5766.419,E2 -5766.419} C_VEL
LIN {X 0,Y 502.869,Z 587.848,A -85,B 0,C 180,E1 -5768.844,E2 -5768.844} C_VEL
LIN {X 0,Y 502.884,Z 587.838,A -85,B 0,C 180,E1 -5772.101,E2 -5772.101} C_VEL
LIN {X 0,Y 502.839,Z 587.846,A -85,B 0,C 180,E1 -5775.4,E2 -5775.4} C_VEL
LIN {X 0,Y 502.837,Z 587.845,A -85,B 0,C 180,E1 -5778.123,E2 -5778.123} C_VEL
LIN {X 0,Y 502.82,Z 587.848,A -85,B 0,C 180,E1 -5780.537,E2 -5780.537} C_VEL
LIN {X 0,Y 502.786,Z 587.856,A -85,B 0,C 180,E1 -5783.041,E2 -5783.041} C_VEL
LIN {X 0,Y 502.834,Z 587.846,A -85,B 0,C 180,E1 -5785.676,E2 -5785.676} C_VEL
LIN {X 0,Y 502.836,Z 587.843,A -85,B 0,C 180,E1 -5788.373,E2 -5788.373} C_VEL
LIN {X 0,Y 502.791,Z 587.853,A -85,B 0,C 180,E1 -5791.501,E2 -5791.501} C_VEL
LIN {X 0,Y 502.801,Z 587.848,A -85,B 0,C 180,E1 -5794.446,E2 -5794.446} C_VEL
LIN {X 0,Y 502.778,Z 587.858,A -85,B 0,C 180,E1 -5797.18,E2 -5797.18} C_VEL
LIN {X 0,Y 502.784,Z 587.852,A -85,B 0,C 180,E1 -5800.016,E2 -5800.016} C_VEL
LIN {X 0,Y 502.799,Z 587.85,A -85,B 0,C 180,E1 -5802.2,E2 -5802.2} C_VEL
LIN {X 0,Y 502.797,Z 587.857,A -85,B 0,C 180,E1 -5805.469,E2 -5805.469} C_VEL
LIN {X 0,Y 502.824,Z 587.849,A -85,B 0,C 180,E1 -5809.005,E2 -5809.005} C_VEL
LIN {X 0,Y 502.793,Z 587.854,A -85,B 0,C 180,E1 -5812.047,E2 -5812.047} C_VEL
LIN {X 0,Y 502.809,Z 587.851,A -85,B 0,C 180,E1 -5815.036,E2 -5815.036} C_VEL
LIN {X 0,Y 502.784,Z 587.857,A -85,B 0,C 180,E1 -5817.916,E2 -5817.916} C_VEL
LIN {X 0,Y 502.824,Z 587.849,A -85,B 0,C 180,E1 -5820.713,E2 -5820.713} C_VEL
LIN {X 0,Y 502.879,Z 587.848,A -85,B 0,C 180,E1 -5824.105,E2 -5824.105} C_VEL
LIN {X 0,Y 502.88,Z 587.903,A -85,B 0,C 180,E1 -5824.327,E2 -5824.327} C_VEL
LIN {X 0,Y 504.814,Z 598.796,A -85,B 0,C 180,E1 -5826.189,E2 -5826.189} C_VEL
LIN {X 0,Y 504.325,Z 614.999,A -85,B 0,C 180,E1 -5828.758,E2 -5828.758} C_VEL
LIN {X 0,Y 503.733,Z 636.634,A -85,B 0,C 180,E1 -5832.126,E2 -5832.126} C_VEL
LIN {X 0,Y 503.355,Z 650.073,A -85,B 0,C 180,E1 -5834.196,E2 -5834.196} C_VEL
LIN {X 0,Y 505.315,Z 664.563,A -85,B 0,C 180,E1 -5834.474,E2 -5834.474} C_VEL
LIN {X 0,Y 504.83,Z 758.971,A -85,B 0,C 180,E1 -5835.848,E2 -5835.848} C_VEL
LIN {X 0,Y 504.565,Z 772.179,A -85,B 0,C 180,E1 -5836.2,E2 -5836.2} C_VEL
LIN {X 0,Y 504.246,Z 784.901,A -85,B 0,C 180,E1 -5836.705,E2 -5836.705} C_VEL
LIN {X 0,Y 503.919,Z 797.153,A -85,B 0,C 180,E1 -5837.371,E2 -5837.371} C_VEL
LIN {X 0,Y 503.525,Z 809.226,A -85,B 0,C 180,E1 -5838.222,E2 -5838.222} C_VEL
LIN {X 0,Y 503.167,Z 819.523,A -85,B 0,C 180,E1 -5839.131,E2 -5839.131} C_VEL
LIN {X 0,Y 502.877,Z 828.778,A -85,B 0,C 180,E1 -5840.143,E2 -5840.143} C_VEL
LIN {X 0,Y 502.606,Z 837.79,A -85,B 0,C 180,E1 -5841.355,E2 -5841.355} C_VEL
LIN {X 0,Y 502.355,Z 845.046,A -85,B 0,C 180,E1 -5842.565,E2 -5842.565} C_VEL
LIN {X 0,Y 502.236,Z 849.941,A -85,B 0,C 180,E1 -5843.573,E2 -5843.573} C_VEL
LIN {X 0,Y 502.183,Z 854.703,A -85,B 0,C 180,E1 -5844.781,E2 -5844.781} C_VEL
LIN {X 0,Y 502.151,Z 858.341,A -85,B 0,C 180,E1 -5845.987,E2 -5845.987} C_VEL
LIN {X 0,Y 502.121,Z 860.219,A -85,B 0,C 180,E1 -5846.791,E2 -5846.791} C_VEL
LIN {X 0,Y 502.12,Z 861.627,A -85,B 0,C 180,E1 -5847.594,E2 -5847.594} C_VEL
LIN {X 0,Y 501.99,Z 863.239,A -85,B 0,C 180,E1 -5849.198,E2 -5849.198} C_VEL
LIN {X 0,Y 501.98,Z 863.46,A -85,B 0,C 180,E1 -5850,E2 -5850} C_VEL
LIN {X 0,Y 502.036,Z 862.637,A -85,B 0,C 180,E1 -5851.604,E2 -5851.604} C_VEL
LIN {X 0,Y 502.12,Z 861.642,A -85,B 0,C 180,E1 -5852.406,E2 -5852.406} C_VEL
LIN {X 0,Y 502.121,Z 860.239,A -85,B 0,C 180,E1 -5853.209,E2 -5853.209} C_VEL
LIN {X 0,Y 502.123,Z 857.287,A -85,B 0,C 180,E1 -5854.415,E2 -5854.415} C_VEL
LIN {X 0,Y 502.238,Z 853.294,A -85,B 0,C 180,E1 -5855.621,E2 -5855.621} C_VEL
LIN {X 0,Y 502.334,Z 847.248,A -85,B 0,C 180,E1 -5857.011,E2 -5857.011} C_VEL
LIN {X 0,Y 502.516,Z 840.431,A -85,B 0,C 180,E1 -5858.242,E2 -5858.242} C_VEL
LIN {X 0,Y 502.754,Z 832.099,A -85,B 0,C 180,E1 -5859.454,E2 -5859.454} C_VEL
LIN {X 0,Y 503.012,Z 823.551,A -85,B 0,C 180,E1 -5860.465,E2 -5860.465} C_VEL
LIN {X 0,Y 503.442,Z 812.997,A -85,B 0,C 180,E1 -5861.474,E2 -5861.474} C_VEL
LIN {X 0,Y 503.729,Z 801.375,A -85,B 0,C 180,E1 -5862.368,E2 -5862.368} C_VEL
LIN {X 0,Y 504.123,Z 789.125,A -85,B 0,C 180,E1 -5863.093,E2 -5863.093} C_VEL
LIN {X 0,Y 504.448,Z 776.656,A -85,B 0,C 180,E1 -5863.649,E2 -5863.649} C_VEL
LIN {X 0,Y 504.753,Z 763.764,A -85,B 0,C 180,E1 -5864.051,E2 -5864.051} C_VEL
LIN {X 0,Y 504.927,Z 748.317,A -85,B 0,C 180,E1 -5864.329,E2 -5864.329} C_VEL
LIN {X 0,Y 505.213,Z 662.561,A -85,B 0,C 180,E1 -5865.562,E2 -5865.562} C_VEL
LIN {X 0,Y 503.38,Z 650.289,A -85,B 0,C 180,E1 -5865.813,E2 -5865.813} C_VEL
LIN {X 0,Y 503.978,Z 628.957,A -85,B 0,C 180,E1 -5869.129,E2 -5869.129} C_VEL
LIN {X 0,Y 504.552,Z 610.062,A -85,B 0,C 180,E1 -5872.091,E2 -5872.091} C_VEL
LIN {X 0,Y 504.916,Z 599.282,A -85,B 0,C 180,E1 -5873.806,E2 -5873.806} C_VEL
LIN {X 0,Y 503.519,Z 590.947,A -85,B 0,C 180,E1 -5875.234,E2 -5875.234} C_VEL
LIN {X 0,Y 502.887,Z 587.846,A -85,B 0,C 180,E1 -5875.783,E2 -5875.783} C_VEL
LIN {X 0,Y 502.841,Z 587.852,A -85,B 0,C 180,E1 -5878.372,E2 -5878.372} C_VEL
LIN {X 0,Y 502.793,Z 587.851,A -85,B 0,C 180,E1 -5881.498,E2 -5881.498} C_VEL
LIN {X 0,Y 502.806,Z 587.857,A -85,B 0,C 180,E1 -5884.444,E2 -5884.444} C_VEL
LIN {X 0,Y 502.78,Z 587.852,A -85,B 0,C 180,E1 -5887.178,E2 -5887.178} C_VEL
LIN {X 0,Y 502.819,Z 587.848,A -85,B 0,C 180,E1 -5890.011,E2 -5890.011} C_VEL
LIN {X 0,Y 502.77,Z 587.854,A -85,B 0,C 180,E1 -5893.23,E2 -5893.23} C_VEL
LIN {X 0,Y 502.786,Z 587.85,A -85,B 0,C 180,E1 -5895.66,E2 -5895.66} C_VEL
LIN {X 0,Y 502.816,Z 587.852,A -85,B 0,C 180,E1 -5898.933,E2 -5898.933} C_VEL
LIN {X 0,Y 502.791,Z 587.85,A -85,B 0,C 180,E1 -5902.045,E2 -5902.045} C_VEL
LIN {X 0,Y 502.804,Z 587.854,A -85,B 0,C 180,E1 -5905.034,E2 -5905.034} C_VEL
LIN {X 0,Y 502.781,Z 587.851,A -85,B 0,C 180,E1 -5907.915,E2 -5907.915} C_VEL
LIN {X 0,Y 502.832,Z 587.85,A -85,B 0,C 180,E1 -5910.712,E2 -5910.712} C_VEL
LIN {X 0,Y 502.874,Z 587.842,A -85,B 0,C 180,E1 -5913.434,E2 -5913.434} C_VEL
LIN {X 0,Y 502.784,Z 587.85,A -85,B 0,C 180,E1 -5916.085,E2 -5916.085} C_VEL
LIN {X 0,Y 502.775,Z 587.855,A -85,B 0,C 180,E1 -5918.688,E2 -5918.688} C_VEL
LIN {X 0,Y 502.822,Z 587.853,A -85,B 0,C 180,E1 -5921.248,E2 -5921.248} C_VEL
LIN {X 0,Y 502.814,Z 587.848,A -85,B 0,C 180,E1 -5923.766,E2 -5923.766} C_VEL
LIN {X 0,Y 502.822,Z 587.846,A -85,B 0,C 180,E1 -5926.254,E2 -5926.254} C_VEL
LIN {X 0,Y 502.872,Z 587.841,A -85,B 0,C 180,E1 -5928.716,E2 -5928.716} C_VEL
LIN {X 0,Y 502.893,Z 587.838,A -85,B 0,C 180,E1 -5931.966,E2 -5931.966} C_VEL
LIN {X 0,Y 502.941,Z 587.831,A -85,B 0,C 180,E1 -5934.386,E2 -5934.386} C_VEL
LIN {X 0,Y 503.015,Z 587.828,A -85,B 0,C 180,E1 -5937.597,E2 -5937.597} C_VEL
LIN {X 0,Y 503.016,Z 587.823,A -85,B 0,C 180,E1 -5940,E2 -5940} C_VEL
LIN {X 0,Y 503.015,Z 587.822,A -85,B 0,C 180,E1 -5942.402,E2 -5942.402} C_VEL
LIN {X 0,Y 502.949,Z 587.839,A -85,B 0,C 180,E1 -5945.613,E2 -5945.613} C_VEL
LIN {X 0,Y 502.892,Z 587.84,A -85,B 0,C 180,E1 -5948.033,E2 -5948.033} C_VEL
LIN {X 0,Y 502.871,Z 587.843,A -85,B 0,C 180,E1 -5951.283,E2 -5951.283} C_VEL
LIN {X 0,Y 502.834,Z 587.844,A -85,B 0,C 180,E1 -5954.571,E2 -5954.571} C_VEL
LIN {X 0,Y 502.851,Z 587.849,A -85,B 0,C 180,E1 -5957.907,E2 -5957.907} C_VEL
LIN {X 0,Y 502.817,Z 587.847,A -85,B 0,C 180,E1 -5960.536,E2 -5960.536} C_VEL
LIN {X 0,Y 502.783,Z 587.851,A -85,B 0,C 180,E1 -5963.04,E2 -5963.04} C_VEL
LIN {X 0,Y 502.831,Z 587.85,A -85,B 0,C 180,E1 -5965.676,E2 -5965.676} C_VEL
LIN {X 0,Y 502.832,Z 587.848,A -85,B 0,C 180,E1 -5968.373,E2 -5968.373} C_VEL
LIN {X 0,Y 502.787,Z 587.852,A -85,B 0,C 180,E1 -5971.5,E2 -5971.5} C_VEL
LIN {X 0,Y 502.796,Z 587.853,A -85,B 0,C 180,E1 -5974.445,E2 -5974.445} C_VEL
LIN {X 0,Y 502.772,Z 587.852,A -85,B 0,C 180,E1 -5977.179,E2 -5977.179} C_VEL
LIN {X 0,Y 502.826,Z 587.852,A -85,B 0,C 180,E1 -5980.011,E2 -5980.011} C_VEL
LIN {X 0,Y 502.819,Z 587.856,A -85,B 0,C 180,E1 -5982.203,E2 -5982.203} C_VEL
LIN {X 0,Y 502.792,Z 587.85,A -85,B 0,C 180,E1 -5985.469,E2 -5985.469} C_VEL
LIN {X 0,Y 502.822,Z 587.849,A -85,B 0,C 180,E1 -5987.865,E2 -5987.865} C_VEL
LIN {X 0,Y 502.795,Z 587.85,A -85,B 0,C 180,E1 -5991.025,E2 -5991.025} C_VEL
LIN {X 0,Y 502.779,Z 587.856,A -85,B 0,C 180,E1 -5994.168,E2 -5994.168} C_VEL
LIN {X 0,Y 502.803,Z 587.849,A -85,B 0,C 180,E1 -5997.235,E2 -5997.235} C_VEL
LIN {X 0,Y 502.103,Z 587.938,A -85,B 0,C 180,E1 -5997.904,E2 -5997.904} C_VEL
LIN {X 0,Y 499.238,Z 588.295,A -85,B 0,C 180,E1 -5998.989,E2 -5998.989} C_VEL
LIN {X 0,Y 496.842,Z 588.594,A -85,B 0,C 180,E1 -5999.864,E2 -5999.864} C_VEL
LIN {X 0,Y 495.825,Z 588.727,A -85,B 0,C 180,E1 -6000.54,E2 -6000.54} C_VEL
LIN {X 0,Y 495.748,Z 588.728,A -85,B 0,C 180,E1 -6000.769,E2 -6000.769} C_VEL
LIN {X 0,Y 495.786,Z 588.723,A -85,B 0,C 180,E1 -6003.933,E2 -6003.933} C_VEL
LIN {X 0,Y 495.761,Z 588.728,A -85,B 0,C 180,E1 -6007.138,E2 -6007.138} C_VEL
LIN {X 0,Y 495.774,Z 588.725,A -85,B 0,C 180,E1 -6010.11,E2 -6010.11} C_VEL
LIN {X 0,Y 495.785,Z 588.73,A -85,B 0,C 180,E1 -6012.682,E2 -6012.682} C_VEL
LIN {X 0,Y 495.787,Z 588.726,A -85,B 0,C 180,E1 -6015.217,E2 -6015.217} C_VEL
LIN {X 0,Y 495.848,Z 588.719,A -85,B 0,C 180,E1 -6018.555,E2 -6018.555} C_VEL
LIN {X 0,Y 495.87,Z 588.712,A -85,B 0,C 180,E1 -6021.852,E2 -6021.852} C_VEL
LIN {X 0,Y 495.887,Z 588.711,A -85,B 0,C 180,E1 -6024.307,E2 -6024.307} C_VEL
LIN {X 0,Y 495.992,Z 588.699,A -85,B 0,C 180,E1 -6027.564,E2 -6027.564} C_VEL
LIN {X 0,Y 495.996,Z 588.696,A -85,B 0,C 180,E1 -6030,E2 -6030} C_VEL
LIN {X 0,Y 495.992,Z 588.697,A -85,B 0,C 180,E1 -6032.436,E2 -6032.436} C_VEL
LIN {X 0,Y 495.887,Z 588.712,A -85,B 0,C 180,E1 -6035.693,E2 -6035.693} C_VEL
LIN {X 0,Y 495.87,Z 588.712,A -85,B 0,C 180,E1 -6038.148,E2 -6038.148} C_VEL
LIN {X 0,Y 495.848,Z 588.721,A -85,B 0,C 180,E1 -6041.445,E2 -6041.445} C_VEL
LIN {X 0,Y 495.787,Z 588.724,A -85,B 0,C 180,E1 -6044.783,E2 -6044.783} C_VEL
LIN {X 0,Y 495.785,Z 588.731,A -85,B 0,C 180,E1 -6047.318,E2 -6047.318} C_VEL
LIN {X 0,Y 495.774,Z 588.729,A -85,B 0,C 180,E1 -6049.89,E2 -6049.89} C_VEL
LIN {X 0,Y 495.76,Z 588.729,A -85,B 0,C 180,E1 -6052.862,E2 -6052.862} C_VEL
LIN {X 0,Y 495.878,Z 588.837,A -85,B 0,C 180,E1 -6055.442,E2 -6055.442} C_VEL
LIN {X 0,Y 496.54,Z 594.396,A -85,B 0,C 180,E1 -6056.68,E2 -6056.68} C_VEL
LIN {X 0,Y 496.271,Z 605.463,A -85,B 0,C 180,E1 -6059.043,E2 -6059.043} C_VEL
LIN {X 0,Y 498.576,Z 617.38,A -85,B 0,C 180,E1 -6059.3,E2 -6059.3} C_VEL
LIN {X 0,Y 497.961,Z 712.328,A -85,B 0,C 180,E1 -6060.711,E2 -6060.711} C_VEL
LIN {X 0,Y 497.695,Z 726.138,A -85,B 0,C 180,E1 -6061.098,E2 -6061.098} C_VEL
LIN {X 0,Y 497.454,Z 738.176,A -85,B 0,C 180,E1 -6061.6,E2 -6061.6} C_VEL
LIN {X 0,Y 497.09,Z 750.303,A -85,B 0,C 180,E1 -6062.281,E2 -6062.281} C_VEL
LIN {X 0,Y 496.669,Z 761.604,A -85,B 0,C 180,E1 -6063.099,E2 -6063.099} C_VEL
LIN {X 0,Y 496.336,Z 771.649,A -85,B 0,C 180,E1 -6064.007,E2 -6064.007} C_VEL
LIN {X 0,Y 495.935,Z 781.414,A -85,B 0,C 180,E1 -6065.102,E2 -6065.102} C_VEL
LIN {X 0,Y 495.649,Z 789.928,A -85,B 0,C 180,E1 -6066.286,E2 -6066.286} C_VEL
LIN {X 0,Y 495.374,Z 797.468,A -85,B 0,C 180,E1 -6067.592,E2 -6067.592} C_VEL
LIN {X 0,Y 495.251,Z 802.564,A -85,B 0,C 180,E1 -6068.695,E2 -6068.695} C_VEL
LIN {X 0,Y 495.127,Z 807.211,A -85,B 0,C 180,E1 -6069.961,E2 -6069.961} C_VEL
LIN {X 0,Y 495.052,Z 810.651,A -85,B 0,C 180,E1 -6071.201,E2 -6071.201} C_VEL
LIN {X 0,Y 494.982,Z 813.034,A -85,B 0,C 180,E1 -6072.412,E2 -6072.412} C_VEL
LIN {X 0,Y 494.924,Z 814.817,A -85,B 0,C 180,E1 -6074.09,E2 -6074.09} C_VEL
LIN {X 0,Y 494.914,Z 815.085,A -85,B 0,C 180,E1 -6075.235,E2 -6075.235} C_VEL
LIN {X 0,Y 494.943,Z 814.573,A -85,B 0,C 180,E1 -6076.399,E2 -6076.399} C_VEL
LIN {X 0,Y 494.981,Z 813.195,A -85,B 0,C 180,E1 -6077.587,E2 -6077.587} C_VEL
LIN {X 0,Y 495.058,Z 809.828,A -85,B 0,C 180,E1 -6079.23,E2 -6079.23} C_VEL
LIN {X 0,Y 495.134,Z 806.686,A -85,B 0,C 180,E1 -6080.303,E2 -6080.303} C_VEL
LIN {X 0,Y 495.306,Z 801.617,A -85,B 0,C 180,E1 -6081.628,E2 -6081.628} C_VEL
LIN {X 0,Y 495.491,Z 794.72,A -85,B 0,C 180,E1 -6083.025,E2 -6083.025} C_VEL
LIN {X 0,Y 495.742,Z 787.432,A -85,B 0,C 180,E1 -6084.194,E2 -6084.194} C_VEL
LIN {X 0,Y 496.072,Z 779.331,A -85,B 0,C 180,E1 -6085.253,E2 -6085.253} C_VEL
LIN {X 0,Y 496.418,Z 768.862,A -85,B 0,C 180,E1 -6086.365,E2 -6086.365} C_VEL
LIN {X 0,Y 496.806,Z 758.562,A -85,B 0,C 180,E1 -6087.242,E2 -6087.242} C_VEL
LIN {X 0,Y 497.224,Z 747.331,A -85,B 0,C 180,E1 -6088,E2 -6088} C_VEL
LIN {X 0,Y 497.492,Z 735.814,A -85,B 0,C 180,E1 -6088.606,E2 -6088.606} C_VEL
LIN {X 0,Y 497.774,Z 722.724,A -85,B 0,C 180,E1 -6089.111,E2 -6089.111} C_VEL
LIN {X 0,Y 497.968,Z 710.49,A -85,B 0,C 180,E1 -6089.417,E2 -6089.417} C_VEL
LIN {X 0,Y 498.509,Z 617.122,A -85,B 0,C 180,E1 -6090.801,E2 -6090.801} C_VEL
LIN {X 0,Y 496.284,Z 605.704,A -85,B 0,C 180,E1 -6091.057,E2 -6091.057} C_VEL
LIN {X 0,Y 496.612,Z 594.306,A -85,B 0,C 180,E1 -6093.53,E2 -6093.53} C_VEL
LIN {X 0,Y 495.799,Z 588.73,A -85,B 0,C 180,E1 -6094.834,E2 -6094.834} C_VEL
LIN {X 0,Y 495.743,Z 588.731,A -85,B 0,C 180,E1 -6097.495,E2 -6097.495} C_VEL
LIN {X 0,Y 495.768,Z 588.729,A -85,B 0,C 180,E1 -6100.11,E2 -6100.11} C_VEL
LIN {X 0,Y 495.778,Z 588.732,A -85,B 0,C 180,E1 -6102.682,E2 -6102.682} C_VEL
LIN {X 0,Y 495.779,Z 588.727,A -85,B 0,C 180,E1 -6105.217,E2 -6105.217} C_VEL
LIN {X 0,Y 495.865,Z 588.721,A -85,B 0,C 180,E1 -6108.556,E2 -6108.556} C_VEL
LIN {X 0,Y 495.864,Z 588.715,A -85,B 0,C 180,E1 -6111.852,E2 -6111.852} C_VEL
LIN {X 0,Y 495.907,Z 588.711,A -85,B 0,C 180,E1 -6114.307,E2 -6114.307} C_VEL
LIN {X 0,Y 495.989,Z 588.699,A -85,B 0,C 180,E1 -6117.564,E2 -6117.564} C_VEL
LIN {X 0,Y 495.987,Z 588.699,A -85,B 0,C 180,E1 -6120,E2 -6120} C_VEL
LIN {X 0,Y 495.985,Z 588.701,A -85,B 0,C 180,E1 -6122.437,E2 -6122.437} C_VEL
LIN {X 0,Y 495.908,Z 588.708,A -85,B 0,C 180,E1 -6125.694,E2 -6125.694} C_VEL
LIN {X 0,Y 495.864,Z 588.714,A -85,B 0,C 180,E1 -6128.148,E2 -6128.148} C_VEL
LIN {X 0,Y 495.868,Z 588.716,A -85,B 0,C 180,E1 -6131.445,E2 -6131.445} C_VEL
LIN {X 0,Y 495.781,Z 588.729,A -85,B 0,C 180,E1 -6134.784,E2 -6134.784} C_VEL
LIN {X 0,Y 495.78,Z 588.73,A -85,B 0,C 180,E1 -6137.319,E2 -6137.319} C_VEL
LIN {X 0,Y 495.77,Z 588.725,A -85,B 0,C 180,E1 -6139.891,E2 -6139.891} C_VEL
LIN {X 0,Y 495.753,Z 588.73,A -85,B 0,C 180,E1 -6142.862,E2 -6142.862} C_VEL
LIN {X 0,Y 495.792,Z 588.72,A -85,B 0,C 180,E1 -6146.068,E2 -6146.068} C_VEL
LIN {X 0,Y 495.774,Z 588.726,A -85,B 0,C 180,E1 -6148.815,E2 -6148.815} C_VEL
LIN {X 0,Y 495.753,Z 588.727,A -85,B 0,C 180,E1 -6151.727,E2 -6151.727} C_VEL
LIN {X 0,Y 495.771,Z 588.725,A -85,B 0,C 180,E1 -6154.696,E2 -6154.696} C_VEL
LIN {X 0,Y 495.729,Z 588.734,A -85,B 0,C 180,E1 -6157.562,E2 -6157.562} C_VEL
LIN {X 0,Y 495.763,Z 588.726,A -85,B 0,C 180,E1 -6160.701,E2 -6160.701} C_VEL
LIN {X 0,Y 495.731,Z 588.736,A -85,B 0,C 180,E1 -6163.696,E2 -6163.696} C_VEL
LIN {X 0,Y 495.726,Z 588.732,A -85,B 0,C 180,E1 -6166.306,E2 -6166.306} C_VEL
LIN {X 0,Y 495.777,Z 588.731,A -85,B 0,C 180,E1 -6169.302,E2 -6169.302} C_VEL
LIN {X 0,Y 495.73,Z 588.731,A -85,B 0,C 180,E1 -6172.44,E2 -6172.44} C_VEL
LIN {X 0,Y 495.784,Z 588.731,A -85,B 0,C 180,E1 -6175.458,E2 -6175.458} C_VEL
LIN {X 0,Y 495.756,Z 588.728,A -85,B 0,C 180,E1 -6178.365,E2 -6178.365} C_VEL
LIN {X 0,Y 495.788,Z 588.731,A -85,B 0,C 180,E1 -6181.508,E2 -6181.508} C_VEL
LIN {X 0,Y 495.854,Z 588.787,A -85,B 0,C 180,E1 -6184.134,E2 -6184.134} C_VEL
LIN {X 0,Y 497.843,Z 599.787,A -85,B 0,C 180,E1 -6186.052,E2 -6186.052} C_VEL
LIN {X 0,Y 497.425,Z 614.651,A -85,B 0,C 180,E1 -6188.448,E2 -6188.448} C_VEL
LIN {X 0,Y 496.753,Z 635.167,A -85,B 0,C 180,E1 -6191.696,E2 -6191.696} C_VEL
LIN {X 0,Y 496.335,Z 649.77,A -85,B 0,C 180,E1 -6193.969,E2 -6193.969} C_VEL
LIN {X 0,Y 498.478,Z 663.888,A -85,B 0,C 180,E1 -6194.251,E2 -6194.251} C_VEL
LIN {X 0,Y 497.922,Z 758.339,A -85,B 0,C 180,E1 -6195.648,E2 -6195.648} C_VEL
LIN {X 0,Y 497.661,Z 771.629,A -85,B 0,C 180,E1 -6196.005,E2 -6196.005} C_VEL
LIN {X 0,Y 497.335,Z 784.398,A -85,B 0,C 180,E1 -6196.517,E2 -6196.517} C_VEL
LIN {X 0,Y 497,Z 795.308,A -85,B 0,C 180,E1 -6197.104,E2 -6197.104} C_VEL
LIN {X 0,Y 496.631,Z 806.181,A -85,B 0,C 180,E1 -6197.849,E2 -6197.849} C_VEL
LIN {X 0,Y 496.247,Z 816.956,A -85,B 0,C 180,E1 -6198.771,E2 -6198.771} C_VEL
LIN {X 0,Y 495.881,Z 826.667,A -85,B 0,C 180,E1 -6199.796,E2 -6199.796} C_VEL
LIN {X 0,Y 495.615,Z 834.63,A -85,B 0,C 180,E1 -6200.821,E2 -6200.821} C_VEL
LIN {X 0,Y 495.359,Z 842.407,A -85,B 0,C 180,E1 -6202.049,E2 -6202.049} C_VEL
LIN {X 0,Y 495.254,Z 847.735,A -85,B 0,C 180,E1 -6203.072,E2 -6203.072} C_VEL
LIN {X 0,Y 495.154,Z 852.898,A -85,B 0,C 180,E1 -6204.298,E2 -6204.298} C_VEL
LIN {X 0,Y 495.025,Z 856.903,A -85,B 0,C 180,E1 -6205.522,E2 -6205.522} C_VEL
LIN {X 0,Y 495.043,Z 859.866,A -85,B 0,C 180,E1 -6206.745,E2 -6206.745} C_VEL
LIN {X 0,Y 495.024,Z 861.276,A -85,B 0,C 180,E1 -6207.559,E2 -6207.559} C_VEL
LIN {X 0,Y 494.911,Z 862.895,A -85,B 0,C 180,E1 -6209.186,E2 -6209.186} C_VEL
LIN {X 0,Y 494.898,Z 863.117,A -85,B 0,C 180,E1 -6210,E2 -6210} C_VEL
LIN {X 0,Y 494.963,Z 862.296,A -85,B 0,C 180,E1 -6211.627,E2 -6211.627} C_VEL
LIN {X 0,Y 495.024,Z 861.299,A -85,B 0,C 180,E1 -6212.441,E2 -6212.441} C_VEL
LIN {X 0,Y 495.043,Z 859.896,A -85,B 0,C 180,E1 -6213.255,E2 -6213.255} C_VEL
LIN {X 0,Y 495.025,Z 856.941,A -85,B 0,C 180,E1 -6214.478,E2 -6214.478} C_VEL
LIN {X 0,Y 495.154,Z 852.945,A -85,B 0,C 180,E1 -6215.702,E2 -6215.702} C_VEL
LIN {X 0,Y 495.258,Z 846.79,A -85,B 0,C 180,E1 -6217.133,E2 -6217.133} C_VEL
LIN {X 0,Y 495.458,Z 840.07,A -85,B 0,C 180,E1 -6218.36,E2 -6218.36} C_VEL
LIN {X 0,Y 495.716,Z 831.73,A -85,B 0,C 180,E1 -6219.589,E2 -6219.589} C_VEL
LIN {X 0,Y 496.002,Z 823.171,A -85,B 0,C 180,E1 -6220.614,E2 -6220.614} C_VEL
LIN {X 0,Y 496.452,Z 812.605,A -85,B 0,C 180,E1 -6221.638,E2 -6221.638} C_VEL
LIN {X 0,Y 496.764,Z 801.177,A -85,B 0,C 180,E1 -6222.529,E2 -6222.529} C_VEL
LIN {X 0,Y 497.124,Z 790.661,A -85,B 0,C 180,E1 -6223.177,E2 -6223.177} C_VEL
LIN {X 0,Y 497.509,Z 778.802,A -85,B 0,C 180,E1 -6223.739,E2 -6223.739} C_VEL
LIN {X 0,Y 497.816,Z 766.039,A -85,B 0,C 180,E1 -6224.173,E2 -6224.173} C_VEL
LIN {X 0,Y 498.044,Z 752.896,A -85,B 0,C 180,E1 -6224.453,E2 -6224.453} C_VEL
LIN {X 0,Y 498.452,Z 663.858,A -85,B 0,C 180,E1 -6225.755,E2 -6225.755} C_VEL
LIN {X 0,Y 496.343,Z 650.014,A -85,B 0,C 180,E1 -6226.035,E2 -6226.035} C_VEL
LIN {X 0,Y 496.994,Z 629.971,A -85,B 0,C 180,E1 -6229.194,E2 -6229.194} C_VEL
LIN {X 0,Y 497.674,Z 609.793,A -85,B 0,C 180,E1 -6232.413,E2 -6232.413} C_VEL
LIN {X 0,Y 497.987,Z 600.329,A -85,B 0,C 180,E1 -6233.947,E2 -6233.947} C_VEL
LIN {X 0,Y 495.853,Z 588.722,A -85,B 0,C 180,E1 -6236.007,E2 -6236.007} C_VEL
LIN {X 0,Y 495.772,Z 588.73,A -85,B 0,C 180,E1 -6238.814,E2 -6238.814} C_VEL
LIN {X 0,Y 495.756,Z 588.729,A -85,B 0,C 180,E1 -6241.725,E2 -6241.725} C_VEL
LIN {X 0,Y 495.776,Z 588.729,A -85,B 0,C 180,E1 -6244.694,E2 -6244.694} C_VEL
LIN {X 0,Y 495.73,Z 588.729,A -85,B 0,C 180,E1 -6247.56,E2 -6247.56} C_VEL
LIN {X 0,Y 495.777,Z 588.731,A -85,B 0,C 180,E1 -6250.698,E2 -6250.698} C_VEL
LIN {X 0,Y 495.731,Z 588.73,A -85,B 0,C 180,E1 -6254,E2 -6254} C_VEL
LIN {X 0,Y 495.73,Z 588.732,A -85,B 0,C 180,E1 -6257.117,E2 -6257.117} C_VEL
LIN {X 0,Y 495.755,Z 588.727,A -85,B 0,C 180,E1 -6259.952,E2 -6259.952} C_VEL
LIN {X 0,Y 495.728,Z 588.735,A -85,B 0,C 180,E1 -6262.551,E2 -6262.551} C_VEL
LIN {X 0,Y 495.779,Z 588.724,A -85,B 0,C 180,E1 -6265.456,E2 -6265.456} C_VEL
LIN {X 0,Y 495.753,Z 588.728,A -85,B 0,C 180,E1 -6268.363,E2 -6268.363} C_VEL
LIN {X 0,Y 495.783,Z 588.724,A -85,B 0,C 180,E1 -6271.505,E2 -6271.505} C_VEL
LIN {X 0,Y 495.792,Z 588.721,A -85,B 0,C 180,E1 -6273.932,E2 -6273.932} C_VEL
LIN {X 0,Y 495.753,Z 588.734,A -85,B 0,C 180,E1 -6277.138,E2 -6277.138} C_VEL
LIN {X 0,Y 495.77,Z 588.724,A -85,B 0,C 180,E1 -6280.109,E2 -6280.109} C_VEL
LIN {X 0,Y 495.779,Z 588.726,A -85,B 0,C 180,E1 -6282.681,E2 -6282.681} C_VEL
LIN {X 0,Y 495.78,Z 588.732,A -85,B 0,C 180,E1 -6285.216,E2 -6285.216} C_VEL
LIN {X 0,Y 495.845,Z 588.716,A -85,B 0,C 180,E1 -6288.554,E2 -6288.554} C_VEL
LIN {X 0,Y 495.864,Z 588.714,A -85,B 0,C 180,E1 -6291.851,E2 -6291.851} C_VEL
LIN {X 0,Y 495.897,Z 588.708,A -85,B 0,C 180,E1 -6294.306,E2 -6294.306} C_VEL
LIN {X 0,Y 495.984,Z 588.704,A -85,B 0,C 180,E1 -6297.563,E2 -6297.563} C_VEL
LIN {X 0,Y 495.987,Z 588.699,A -85,B 0,C 180,E1 -6300,E2 -6300} C_VEL
LIN {X 0,Y 495.984,Z 588.697,A -85,B 0,C 180,E1 -6302.436,E2 -6302.436} C_VEL
LIN {X 0,Y 495.903,Z 588.715,A -85,B 0,C 180,E1 -6305.693,E2 -6305.693} C_VEL
LIN {X 0,Y 495.863,Z 588.714,A -85,B 0,C 180,E1 -6308.148,E2 -6308.148} C_VEL
LIN {X 0,Y 495.844,Z 588.721,A -85,B 0,C 180,E1 -6311.445,E2 -6311.445} C_VEL
LIN {X 0,Y 495.779,Z 588.723,A -85,B 0,C 180,E1 -6314.783,E2 -6314.783} C_VEL
LIN {X 0,Y 495.777,Z 588.726,A -85,B 0,C 180,E1 -6317.318,E2 -6317.318} C_VEL
LIN {X 0,Y 495.768,Z 588.733,A -85,B 0,C 180,E1 -6319.89,E2 -6319.89} C_VEL
LIN {X 0,Y 495.75,Z 588.727,A -85,B 0,C 180,E1 -6322.861,E2 -6322.861} C_VEL
LIN {X 0,Y 495.789,Z 588.729,A -85,B 0,C 180,E1 -6326.067,E2 -6326.067} C_VEL
LIN {X 0,Y 495.77,Z 588.724,A -85,B 0,C 180,E1 -6328.814,E2 -6328.814} C_VEL
LIN {X 0,Y 495.749,Z 588.731,A -85,B 0,C 180,E1 -6331.726,E2 -6331.726} C_VEL
LIN {X 0,Y 495.766,Z 588.726,A -85,B 0,C 180,E1 -6334.695,E2 -6334.695} C_VEL
LIN {X 0,Y 495.724,Z 588.732,A -85,B 0,C 180,E1 -6337.562,E2 -6337.562} C_VEL
LIN {X 0,Y 495.792,Z 588.729,A -85,B 0,C 180,E1 -6340.053,E2 -6340.053} C_VEL
LIN {X 0,Y 495.756,Z 588.727,A -85,B 0,C 180,E1 -6342.879,E2 -6342.879} C_VEL
LIN {X 0,Y 495.728,Z 588.734,A -85,B 0,C 180,E1 -6346,E2 -6346} C_VEL
LIN {X 0,Y 495.756,Z 588.73,A -85,B 0,C 180,E1 -6348.706,E2 -6348.706} C_VEL
LIN {X 0,Y 495.744,Z 588.727,A -85,B 0,C 180,E1 -6351.409,E2 -6351.409} C_VEL
LIN {X 0,Y 495.751,Z 588.736,A -85,B 0,C 180,E1 -6354.464,E2 -6354.464} C_VEL
LIN {X 0,Y 495.764,Z 588.725,A -85,B 0,C 180,E1 -6357.406,E2 -6357.406} C_VEL
LIN {X 0,Y 495.761,Z 588.73,A -85,B 0,C 180,E1 -6360.254,E2 -6360.254} C_VEL
LIN {X 0,Y 495.748,Z 588.728,A -85,B 0,C 180,E1 -6360.769,E2 -6360.769} C_VEL
LIN {X 0,Y 495.091,Z 588.812,A -85,B 0,C 180,E1 -6361.448,E2 -6361.448} C_VEL
LIN {X 0,Y 492.234,Z 589.174,A -85,B 0,C 180,E1 -6362.55,E2 -6362.55} C_VEL
LIN {X 0,Y 489.825,Z 589.468,A -85,B 0,C 180,E1 -6363.439,E2 -6363.439} C_VEL
LIN {X 0,Y 488.81,Z 589.594,A -85,B 0,C 180,E1 -6364.125,E2 -6364.125} C_VEL
LIN {X 0,Y 488.738,Z 589.605,A -85,B 0,C 180,E1 -6364.358,E2 -6364.358} C_VEL
LIN {X 0,Y 488.723,Z 589.604,A -85,B 0,C 180,E1 -6367.154,E2 -6367.154} C_VEL
LIN {X 0,Y 488.725,Z 589.602,A -85,B 0,C 180,E1 -6369.811,E2 -6369.811} C_VEL
LIN {X 0,Y 488.732,Z 589.605,A -85,B 0,C 180,E1 -6372.424,E2 -6372.424} C_VEL
LIN {X 0,Y 488.758,Z 589.604,A -85,B 0,C 180,E1 -6375,E2 -6375} C_VEL
LIN {X 0,Y 488.802,Z 589.595,A -85,B 0,C 180,E1 -6378.388,E2 -6378.388} C_VEL
LIN {X 0,Y 488.815,Z 589.591,A -85,B 0,C 180,E1 -6381.734,E2 -6381.734} C_VEL
LIN {X 0,Y 488.845,Z 589.587,A -85,B 0,C 180,E1 -6384.224,E2 -6384.224} C_VEL
LIN {X 0,Y 488.959,Z 589.575,A -85,B 0,C 180,E1 -6387.529,E2 -6387.529} C_VEL
LIN {X 0,Y 488.951,Z 589.579,A -85,B 0,C 180,E1 -6390.824,E2 -6390.824} C_VEL
LIN {X 0,Y 488.96,Z 589.574,A -85,B 0,C 180,E1 -6392.471,E2 -6392.471} C_VEL
LIN {X 0,Y 488.845,Z 589.588,A -85,B 0,C 180,E1 -6395.776,E2 -6395.776} C_VEL
LIN {X 0,Y 488.814,Z 589.591,A -85,B 0,C 180,E1 -6398.266,E2 -6398.266} C_VEL
LIN {X 0,Y 488.802,Z 589.597,A -85,B 0,C 180,E1 -6401.612,E2 -6401.612} C_VEL
LIN {X 0,Y 488.759,Z 589.602,A -85,B 0,C 180,E1 -6405,E2 -6405} C_VEL
LIN {X 0,Y 488.751,Z 589.599,A -85,B 0,C 180,E1 -6408.442,E2 -6408.442} C_VEL
LIN {X 0,Y 488.703,Z 589.61,A -85,B 0,C 180,E1 -6411.07,E2 -6411.07} C_VEL
LIN {X 0,Y 488.689,Z 589.614,A -85,B 0,C 180,E1 -6413.745,E2 -6413.745} C_VEL
LIN {X 0,Y 488.826,Z 589.74,A -85,B 0,C 180,E1 -6415.295,E2 -6415.295} C_VEL
LIN {X 0,Y 489.578,Z 594.696,A -85,B 0,C 180,E1 -6416.423,E2 -6416.423} C_VEL
LIN {X 0,Y 489.295,Z 605.572,A -85,B 0,C 180,E1 -6418.787,E2 -6418.787} C_VEL
LIN {X 0,Y 491.806,Z 618.959,A -85,B 0,C 180,E1 -6419.097,E2 -6419.097} C_VEL
LIN {X 0,Y 491.094,Z 712.726,A -85,B 0,C 180,E1 -6420.514,E2 -6420.514} C_VEL
LIN {X 0,Y 490.826,Z 726.073,A -85,B 0,C 180,E1 -6420.891,E2 -6420.891} C_VEL
LIN {X 0,Y 490.562,Z 738.379,A -85,B 0,C 180,E1 -6421.407,E2 -6421.407} C_VEL
LIN {X 0,Y 490.152,Z 749.673,A -85,B 0,C 180,E1 -6422.04,E2 -6422.04} C_VEL
LIN {X 0,Y 489.77,Z 760.543,A -85,B 0,C 180,E1 -6422.82,E2 -6422.82} C_VEL
LIN {X 0,Y 489.403,Z 771.403,A -85,B 0,C 180,E1 -6423.797,E2 -6423.797} C_VEL
LIN {X 0,Y 489.052,Z 780.269,A -85,B 0,C 180,E1 -6424.779,E2 -6424.779} C_VEL
LIN {X 0,Y 488.712,Z 788.37,A -85,B 0,C 180,E1 -6425.873,E2 -6425.873} C_VEL
LIN {X 0,Y 488.381,Z 796.207,A -85,B 0,C 180,E1 -6427.184,E2 -6427.184} C_VEL
LIN {X 0,Y 488.18,Z 802.904,A -85,B 0,C 180,E1 -6428.607,E2 -6428.607} C_VEL
LIN {X 0,Y 488.058,Z 807.196,A -85,B 0,C 180,E1 -6429.781,E2 -6429.781} C_VEL
LIN {X 0,Y 487.968,Z 810.486,A -85,B 0,C 180,E1 -6430.942,E2 -6430.942} C_VEL
LIN {X 0,Y 487.885,Z 813.707,A -85,B 0,C 180,E1 -6432.611,E2 -6432.611} C_VEL
LIN {X 0,Y 487.842,Z 815.067,A -85,B 0,C 180,E1 -6433.92,E2 -6433.92} C_VEL
LIN {X 0,Y 487.831,Z 815.456,A -85,B 0,C 180,E1 -6435.096,E2 -6435.096} C_VEL
LIN {X 0,Y 487.863,Z 815.031,A -85,B 0,C 180,E1 -6436.254,E2 -6436.254} C_VEL
LIN {X 0,Y 487.884,Z 813.857,A -85,B 0,C 180,E1 -6437.388,E2 -6437.388} C_VEL
LIN {X 0,Y 487.995,Z 810.755,A -85,B 0,C 180,E1 -6439.06,E2 -6439.06} C_VEL
LIN {X 0,Y 488.055,Z 807.56,A -85,B 0,C 180,E1 -6440.218,E2 -6440.218} C_VEL
LIN {X 0,Y 488.178,Z 803.35,A -85,B 0,C 180,E1 -6441.391,E2 -6441.391} C_VEL
LIN {X 0,Y 488.325,Z 798.034,A -85,B 0,C 180,E1 -6442.574,E2 -6442.574} C_VEL
LIN {X 0,Y 488.611,Z 790.781,A -85,B 0,C 180,E1 -6443.863,E2 -6443.863} C_VEL
LIN {X 0,Y 488.923,Z 782.716,A -85,B 0,C 180,E1 -6445.017,E2 -6445.017} C_VEL
LIN {X 0,Y 489.33,Z 773.722,A -85,B 0,C 180,E1 -6446.067,E2 -6446.067} C_VEL
LIN {X 0,Y 489.689,Z 763.247,A -85,B 0,C 180,E1 -6447.062,E2 -6447.062} C_VEL
LIN {X 0,Y 490.144,Z 751.188,A -85,B 0,C 180,E1 -6447.959,E2 -6447.959} C_VEL
LIN {X 0,Y 490.544,Z 739.178,A -85,B 0,C 180,E1 -6448.652,E2 -6448.652} C_VEL
LIN {X 0,Y 490.846,Z 726.248,A -85,B 0,C 180,E1 -6449.197,E2 -6449.197} C_VEL
LIN {X 0,Y 491.058,Z 713.707,A -85,B 0,C 180,E1 -6449.556,E2 -6449.556} C_VEL
LIN {X 0,Y 491.341,Z 679.843,A -85,B 0,C 180,E1 -6450.089,E2 -6450.089} C_VEL
LIN {X 0,Y 491.699,Z 617.976,A -85,B 0,C 180,E1 -6451.017,E2 -6451.017} C_VEL
LIN {X 0,Y 489.357,Z 606.047,A -85,B 0,C 180,E1 -6451.296,E2 -6451.296} C_VEL
LIN {X 0,Y 489.674,Z 595.654,A -85,B 0,C 180,E1 -6453.582,E2 -6453.582} C_VEL
LIN {X 0,Y 488.77,Z 589.605,A -85,B 0,C 180,E1 -6454.978,E2 -6454.978} C_VEL
LIN {X 0,Y 488.69,Z 589.612,A -85,B 0,C 180,E1 -6458.043,E2 -6458.043} C_VEL
LIN {X 0,Y 488.736,Z 589.609,A -85,B 0,C 180,E1 -6460.687,E2 -6460.687} C_VEL
LIN {X 0,Y 488.722,Z 589.605,A -85,B 0,C 180,E1 -6463.286,E2 -6463.286} C_VEL
LIN {X 0,Y 488.73,Z 589.604,A -85,B 0,C 180,E1 -6465.85,E2 -6465.85} C_VEL
LIN {X 0,Y 488.823,Z 589.596,A -85,B 0,C 180,E1 -6468.388,E2 -6468.388} C_VEL
LIN {X 0,Y 488.808,Z 589.594,A -85,B 0,C 180,E1 -6471.734,E2 -6471.734} C_VEL
LIN {X 0,Y 488.863,Z 589.588,A -85,B 0,C 180,E1 -6474.225,E2 -6474.225} C_VEL
LIN {X 0,Y 488.957,Z 589.575,A -85,B 0,C 180,E1 -6477.529,E2 -6477.529} C_VEL
LIN {X 0,Y 488.959,Z 589.574,A -85,B 0,C 180,E1 -6480,E2 -6480} C_VEL
LIN {X 0,Y 488.953,Z 589.577,A -85,B 0,C 180,E1 -6482.472,E2 -6482.472} C_VEL
LIN {X 0,Y 488.864,Z 589.586,A -85,B 0,C 180,E1 -6485.776,E2 -6485.776} C_VEL
LIN {X 0,Y 488.809,Z 589.593,A -85,B 0,C 180,E1 -6488.267,E2 -6488.267} C_VEL
LIN {X 0,Y 488.825,Z 589.591,A -85,B 0,C 180,E1 -6491.612,E2 -6491.612} C_VEL
LIN {X 0,Y 488.753,Z 589.607,A -85,B 0,C 180,E1 -6495.001,E2 -6495.001} C_VEL
LIN {X 0,Y 488.746,Z 589.601,A -85,B 0,C 180,E1 -6498.443,E2 -6498.443} C_VEL
LIN {X 0,Y 488.698,Z 589.614,A -85,B 0,C 180,E1 -6501.072,E2 -6501.072} C_VEL
LIN {X 0,Y 488.685,Z 589.609,A -85,B 0,C 180,E1 -6503.746,E2 -6503.746} C_VEL
LIN {X 0,Y 488.792,Z 589.597,A -85,B 0,C 180,E1 -6506.946,E2 -6506.946} C_VEL
LIN {X 0,Y 488.713,Z 589.603,A -85,B 0,C 180,E1 -6510.366,E2 -6510.366} C_VEL
LIN {X 0,Y 488.73,Z 589.607,A -85,B 0,C 180,E1 -6513.485,E2 -6513.485} C_VEL
LIN {X 0,Y 488.684,Z 589.607,A -85,B 0,C 180,E1 -6516.357,E2 -6516.357} C_VEL
LIN {X 0,Y 488.726,Z 589.608,A -85,B 0,C 180,E1 -6519.252,E2 -6519.252} C_VEL
LIN {X 0,Y 488.691,Z 589.608,A -85,B 0,C 180,E1 -6522.526,E2 -6522.526} C_VEL
LIN {X 0,Y 488.709,Z 589.611,A -85,B 0,C 180,E1 -6525.2,E2 -6525.2} C_VEL
LIN {X 0,Y 488.709,Z 589.606,A -85,B 0,C 180,E1 -6528.401,E2 -6528.401} C_VEL
LIN {X 0,Y 488.739,Z 589.603,A -85,B 0,C 180,E1 -6530.943,E2 -6530.943} C_VEL
LIN {X 0,Y 488.685,Z 589.614,A -85,B 0,C 180,E1 -6533.87,E2 -6533.87} C_VEL
LIN {X 0,Y 488.738,Z 589.605,A -85,B 0,C 180,E1 -6536.878,E2 -6536.878} C_VEL
LIN {X 0,Y 488.724,Z 589.61,A -85,B 0,C 180,E1 -6539.782,E2 -6539.782} C_VEL
LIN {X 0,Y 488.792,Z 589.599,A -85,B 0,C 180,E1 -6543.057,E2 -6543.057} C_VEL
LIN {X 0,Y 488.795,Z 589.672,A -85,B 0,C 180,E1 -6543.933,E2 -6543.933} C_VEL
LIN {X 0,Y 490.899,Z 600.862,A -85,B 0,C 180,E1 -6545.92,E2 -6545.92} C_VEL
LIN {X 0,Y 490.588,Z 612.978,A -85,B 0,C 180,E1 -6547.911,E2 -6547.911} C_VEL
LIN {X 0,Y 489.806,Z 634.551,A -85,B 0,C 180,E1 -6551.388,E2 -6551.388} C_VEL
LIN {X 0,Y 489.352,Z 649.484,A -85,B 0,C 180,E1 -6553.736,E2 -6553.736} C_VEL
LIN {X 0,Y 491.623,Z 665.487,A -85,B 0,C 180,E1 -6554.055,E2 -6554.055} C_VEL
LIN {X 0,Y 491.03,Z 757.697,A -85,B 0,C 180,E1 -6555.442,E2 -6555.442} C_VEL
LIN {X 0,Y 490.767,Z 771.08,A -85,B 0,C 180,E1 -6555.805,E2 -6555.805} C_VEL
LIN {X 0,Y 490.425,Z 783.895,A -85,B 0,C 180,E1 -6556.323,E2 -6556.323} C_VEL
LIN {X 0,Y 490.036,Z 795.148,A -85,B 0,C 180,E1 -6556.936,E2 -6556.936} C_VEL
LIN {X 0,Y 489.599,Z 807.04,A -85,B 0,C 180,E1 -6557.777,E2 -6557.777} C_VEL
LIN {X 0,Y 489.2,Z 817.612,A -85,B 0,C 180,E1 -6558.712,E2 -6558.712} C_VEL
LIN {X 0,Y 488.844,Z 826.255,A -85,B 0,C 180,E1 -6559.647,E2 -6559.647} C_VEL
LIN {X 0,Y 488.556,Z 834.231,A -85,B 0,C 180,E1 -6560.687,E2 -6560.687} C_VEL
LIN {X 0,Y 488.293,Z 842.022,A -85,B 0,C 180,E1 -6561.933,E2 -6561.933} C_VEL
LIN {X 0,Y 488.07,Z 849.195,A -85,B 0,C 180,E1 -6563.385,E2 -6563.385} C_VEL
LIN {X 0,Y 488.052,Z 853.977,A -85,B 0,C 180,E1 -6564.629,E2 -6564.629} C_VEL
LIN {X 0,Y 487.946,Z 857.625,A -85,B 0,C 180,E1 -6565.87,E2 -6565.87} C_VEL
LIN {X 0,Y 487.967,Z 859.514,A -85,B 0,C 180,E1 -6566.697,E2 -6566.697} C_VEL
LIN {X 0,Y 487.932,Z 860.926,A -85,B 0,C 180,E1 -6567.523,E2 -6567.523} C_VEL
LIN {X 0,Y 487.892,Z 861.933,A -85,B 0,C 180,E1 -6568.349,E2 -6568.349} C_VEL
LIN {X 0,Y 487.819,Z 862.774,A -85,B 0,C 180,E1 -6570,E2 -6570} C_VEL
LIN {X 0,Y 487.892,Z 861.954,A -85,B 0,C 180,E1 -6571.651,E2 -6571.651} C_VEL
LIN {X 0,Y 487.932,Z 860.956,A -85,B 0,C 180,E1 -6572.477,E2 -6572.477} C_VEL
LIN {X 0,Y 487.967,Z 859.553,A -85,B 0,C 180,E1 -6573.303,E2 -6573.303} C_VEL
LIN {X 0,Y 487.935,Z 856.595,A -85,B 0,C 180,E1 -6574.544,E2 -6574.544} C_VEL
LIN {X 0,Y 488.05,Z 852.595,A -85,B 0,C 180,E1 -6575.785,E2 -6575.785} C_VEL
LIN {X 0,Y 488.184,Z 846.435,A -85,B 0,C 180,E1 -6577.236,E2 -6577.236} C_VEL
LIN {X 0,Y 488.388,Z 839.707,A -85,B 0,C 180,E1 -6578.482,E2 -6578.482} C_VEL
LIN {X 0,Y 488.655,Z 831.36,A -85,B 0,C 180,E1 -6579.729,E2 -6579.729} C_VEL
LIN {X 0,Y 489.001,Z 822.791,A -85,B 0,C 180,E1 -6580.768,E2 -6580.768} C_VEL
LIN {X 0,Y 489.45,Z 812.212,A -85,B 0,C 180,E1 -6581.807,E2 -6581.807} C_VEL
LIN {X 0,Y 489.759,Z 801.865,A -85,B 0,C 180,E1 -6582.631,E2 -6582.631} C_VEL
LIN {X 0,Y 490.185,Z 790.233,A -85,B 0,C 180,E1 -6583.367,E2 -6583.367} C_VEL
LIN {X 0,Y 490.573,Z 778.335,A -85,B 0,C 180,E1 -6583.937,E2 -6583.937} C_VEL
LIN {X 0,Y 490.928,Z 765.529,A -85,B 0,C 180,E1 -6584.376,E2 -6584.376} C_VEL
LIN {X 0,Y 491.176,Z 752.259,A -85,B 0,C 180,E1 -6584.66,E2 -6584.66} C_VEL
LIN {X 0,Y 491.594,Z 664.594,A -85,B 0,C 180,E1 -6585.964,E2 -6585.964} C_VEL
LIN {X 0,Y 489.371,Z 649.6,A -85,B 0,C 180,E1 -6586.285,E2 -6586.285} C_VEL
LIN {X 0,Y 490.022,Z 629.643,A -85,B 0,C 180,E1 -6589.478,E2 -6589.478} C_VEL
LIN {X 0,Y 490.735,Z 610.85,A -85,B 0,C 180,E1 -6592.525,E2 -6592.525} C_VEL
LIN {X 0,Y 491.047,Z 601.461,A -85,B 0,C 180,E1 -6594.072,E2 -6594.072} C_VEL
LIN {X 0,Y 488.796,Z 589.602,A -85,B 0,C 180,E1 -6596.21,E2 -6596.21} C_VEL
LIN {X 0,Y 488.724,Z 589.605,A -85,B 0,C 180,E1 -6599.27,E2 -6599.27} C_VEL
LIN {X 0,Y 488.703,Z 589.612,A -85,B 0,C 180,E1 -6602.146,E2 -6602.146} C_VEL
LIN {X 0,Y 488.722,Z 589.603,A -85,B 0,C 180,E1 -6605.114,E2 -6605.114} C_VEL
LIN {X 0,Y 488.682,Z 589.612,A -85,B 0,C 180,E1 -6608.199,E2 -6608.199} C_VEL
LIN {X 0,Y 488.747,Z 589.605,A -85,B 0,C 180,E1 -6610.348,E2 -6610.348} C_VEL
LIN {X 0,Y 488.684,Z 589.607,A -85,B 0,C 180,E1 -6613.653,E2 -6613.653} C_VEL
LIN {X 0,Y 488.689,Z 589.611,A -85,B 0,C 180,E1 -6616.345,E2 -6616.345} C_VEL
LIN {X 0,Y 488.715,Z 589.61,A -85,B 0,C 180,E1 -6618.585,E2 -6618.585} C_VEL
LIN {X 0,Y 488.7,Z 589.611,A -85,B 0,C 180,E1 -6620.946,E2 -6620.946} C_VEL
LIN {X 0,Y 488.68,Z 589.607,A -85,B 0,C 180,E1 -6623.868,E2 -6623.868} C_VEL
LIN {X 0,Y 488.733,Z 589.61,A -85,B 0,C 180,E1 -6626.876,E2 -6626.876} C_VEL
LIN {X 0,Y 488.728,Z 589.602,A -85,B 0,C 180,E1 -6629.781,E2 -6629.781} C_VEL
LIN {X 0,Y 488.792,Z 589.601,A -85,B 0,C 180,E1 -6633.054,E2 -6633.054} C_VEL
LIN {X 0,Y 488.685,Z 589.607,A -85,B 0,C 180,E1 -6636.254,E2 -6636.254} C_VEL
LIN {X 0,Y 488.738,Z 589.608,A -85,B 0,C 180,E1 -6639.175,E2 -6639.175} C_VEL
LIN {X 0,Y 488.751,Z 589.601,A -85,B 0,C 180,E1 -6641.627,E2 -6641.627} C_VEL
LIN {X 0,Y 488.752,Z 589.605,A -85,B 0,C 180,E1 -6644.999,E2 -6644.999} C_VEL
LIN {X 0,Y 488.799,Z 589.593,A -85,B 0,C 180,E1 -6648.387,E2 -6648.387} C_VEL
LIN {X 0,Y 488.809,Z 589.594,A -85,B 0,C 180,E1 -6651.733,E2 -6651.733} C_VEL
LIN {X 0,Y 488.855,Z 589.586,A -85,B 0,C 180,E1 -6654.224,E2 -6654.224} C_VEL
LIN {X 0,Y 488.952,Z 589.581,A -85,B 0,C 180,E1 -6657.528,E2 -6657.528} C_VEL
LIN {X 0,Y 488.959,Z 589.575,A -85,B 0,C 180,E1 -6660,E2 -6660} C_VEL
LIN {X 0,Y 488.952,Z 589.573,A -85,B 0,C 180,E1 -6662.471,E2 -6662.471} C_VEL
LIN {X 0,Y 488.86,Z 589.591,A -85,B 0,C 180,E1 -6665.775,E2 -6665.775} C_VEL
LIN {X 0,Y 488.808,Z 589.593,A -85,B 0,C 180,E1 -6668.266,E2 -6668.266} C_VEL
LIN {X 0,Y 488.797,Z 589.601,A -85,B 0,C 180,E1 -6671.612,E2 -6671.612} C_VEL
LIN {X 0,Y 488.751,Z 589.599,A -85,B 0,C 180,E1 -6675,E2 -6675} C_VEL
LIN {X 0,Y 488.744,Z 589.601,A -85,B 0,C 180,E1 -6678.442,E2 -6678.442} C_VEL
LIN {X 0,Y 488.696,Z 589.606,A -85,B 0,C 180,E1 -6681.071,E2 -6681.071} C_VEL
LIN {X 0,Y 488.683,Z 589.614,A -85,B 0,C 180,E1 -6683.745,E2 -6683.745} C_VEL
LIN {X 0,Y 488.789,Z 589.594,A -85,B 0,C 180,E1 -6686.945,E2 -6686.945} C_VEL
LIN {X 0,Y 488.709,Z 589.608,A -85,B 0,C 180,E1 -6690.365,E2 -6690.365} C_VEL
LIN {X 0,Y 488.726,Z 589.603,A -85,B 0,C 180,E1 -6693.485,E2 -6693.485} C_VEL
LIN {X 0,Y 488.68,Z 589.613,A -85,B 0,C 180,E1 -6696.356,E2 -6696.356} C_VEL
LIN {X 0,Y 488.741,Z 589.6,A -85,B 0,C 180,E1 -6699.25,E2 -6699.25} C_VEL
LIN {X 0,Y 488.724,Z 589.603,A -85,B 0,C 180,E1 -6701.604,E2 -6701.604} C_VEL
LIN {X 0,Y 488.694,Z 589.611,A -85,B 0,C 180,E1 -6704.025,E2 -6704.025} C_VEL
LIN {X 0,Y 488.707,Z 589.604,A -85,B 0,C 180,E1 -6707.173,E2 -6707.173} C_VEL
LIN {X 0,Y 488.725,Z 589.603,A -85,B 0,C 180,E1 -6709.677,E2 -6709.677} C_VEL
LIN {X 0,Y 488.676,Z 589.611,A -85,B 0,C 180,E1 -6712.842,E2 -6712.842} C_VEL
LIN {X 0,Y 488.729,Z 589.603,A -85,B 0,C 180,E1 -6715.888,E2 -6715.888} C_VEL
LIN {X 0,Y 488.689,Z 589.611,A -85,B 0,C 180,E1 -6718.821,E2 -6718.821} C_VEL
LIN {X 0,Y 488.739,Z 589.6,A -85,B 0,C 180,E1 -6721.672,E2 -6721.672} C_VEL
LIN {X 0,Y 488.738,Z 589.605,A -85,B 0,C 180,E1 -6724.358,E2 -6724.358} C_VEL
LIN {X 0,Y 488.095,Z 589.691,A -85,B 0,C 180,E1 -6725.045,E2 -6725.045} C_VEL
LIN {X 0,Y 485.227,Z 590.045,A -85,B 0,C 180,E1 -6726.162,E2 -6726.162} C_VEL
LIN {X 0,Y 482.781,Z 590.346,A -85,B 0,C 180,E1 -6727.062,E2 -6727.062} C_VEL
LIN {X 0,Y 481.723,Z 590.474,A -85,B 0,C 180,E1 -6727.757,E2 -6727.757} C_VEL
LIN {X 0,Y 481.634,Z 590.486,A -85,B 0,C 180,E1 -6727.993,E2 -6727.993} C_VEL
LIN {X 0,Y 481.704,Z 590.481,A -85,B 0,C 180,E1 -6730.394,E2 -6730.394} C_VEL
LIN {X 0,Y 481.689,Z 590.483,A -85,B 0,C 180,E1 -6733.034,E2 -6733.034} C_VEL
LIN {X 0,Y 481.688,Z 590.479,A -85,B 0,C 180,E1 -6735.639,E2 -6735.639} C_VEL
LIN {X 0,Y 481.748,Z 590.472,A -85,B 0,C 180,E1 -6738.215,E2 -6738.215} C_VEL
LIN {X 0,Y 481.76,Z 590.47,A -85,B 0,C 180,E1 -6741.612,E2 -6741.612} C_VEL
LIN {X 0,Y 481.805,Z 590.464,A -85,B 0,C 180,E1 -6744.14,E2 -6744.14} C_VEL
LIN {X 0,Y 481.926,Z 590.452,A -85,B 0,C 180,E1 -6747.493,E2 -6747.493} C_VEL
LIN {X 0,Y 481.903,Z 590.457,A -85,B 0,C 180,E1 -6750.836,E2 -6750.836} C_VEL
LIN {X 0,Y 481.926,Z 590.45,A -85,B 0,C 180,E1 -6752.507,E2 -6752.507} C_VEL
LIN {X 0,Y 481.805,Z 590.465,A -85,B 0,C 180,E1 -6755.86,E2 -6755.86} C_VEL
LIN {X 0,Y 481.76,Z 590.47,A -85,B 0,C 180,E1 -6758.388,E2 -6758.388} C_VEL
LIN {X 0,Y 481.747,Z 590.473,A -85,B 0,C 180,E1 -6761.785,E2 -6761.785} C_VEL
LIN {X 0,Y 481.739,Z 590.479,A -85,B 0,C 180,E1 -6765.224,E2 -6765.224} C_VEL
LIN {X 0,Y 481.709,Z 590.477,A -85,B 0,C 180,E1 -6768.721,E2 -6768.721} C_VEL
LIN {X 0,Y 481.643,Z 590.493,A -85,B 0,C 180,E1 -6771.394,E2 -6771.394} C_VEL
LIN {X 0,Y 481.68,Z 590.486,A -85,B 0,C 180,E1 -6774.112,E2 -6774.112} C_VEL
LIN {X 0,Y 481.762,Z 590.676,A -85,B 0,C 180,E1 -6775.152,E2 -6775.152} C_VEL
LIN {X 0,Y 482.596,Z 595.937,A -85,B 0,C 180,E1 -6776.369,E2 -6776.369} C_VEL
LIN {X 0,Y 482.317,Z 605.926,A -85,B 0,C 180,E1 -6778.562,E2 -6778.562} C_VEL
LIN {X 0,Y 485.003,Z 619.896,A -85,B 0,C 180,E1 -6778.878,E2 -6778.878} C_VEL
LIN {X 0,Y 484.221,Z 712.172,A -85,B 0,C 180,E1 -6780.288,E2 -6780.288} C_VEL
LIN {X 0,Y 483.966,Z 725.744,A -85,B 0,C 180,E1 -6780.669,E2 -6780.669} C_VEL
LIN {X 0,Y 483.68,Z 737.944,A -85,B 0,C 180,E1 -6781.178,E2 -6781.178} C_VEL
LIN {X 0,Y 483.259,Z 749.363,A -85,B 0,C 180,E1 -6781.814,E2 -6781.814} C_VEL
LIN {X 0,Y 482.863,Z 760.074,A -85,B 0,C 180,E1 -6782.583,E2 -6782.583} C_VEL
LIN {X 0,Y 482.421,Z 771.49,A -85,B 0,C 180,E1 -6783.613,E2 -6783.613} C_VEL
LIN {X 0,Y 482.044,Z 780.75,A -85,B 0,C 180,E1 -6784.652,E2 -6784.652} C_VEL
LIN {X 0,Y 481.716,Z 788.43,A -85,B 0,C 180,E1 -6785.702,E2 -6785.702} C_VEL
LIN {X 0,Y 481.365,Z 796.311,A -85,B 0,C 180,E1 -6787.031,E2 -6787.031} C_VEL
LIN {X 0,Y 481.151,Z 802.734,A -85,B 0,C 180,E1 -6788.396,E2 -6788.396} C_VEL
LIN {X 0,Y 481.007,Z 807.184,A -85,B 0,C 180,E1 -6789.602,E2 -6789.602} C_VEL
LIN {X 0,Y 480.887,Z 811.387,A -85,B 0,C 180,E1 -6791.12,E2 -6791.12} C_VEL
LIN {X 0,Y 480.802,Z 813.569,A -85,B 0,C 180,E1 -6792.251,E2 -6792.251} C_VEL
LIN {X 0,Y 480.762,Z 815.004,A -85,B 0,C 180,E1 -6793.397,E2 -6793.397} C_VEL
LIN {X 0,Y 480.749,Z 815.714,A -85,B 0,C 180,E1 -6794.563,E2 -6794.563} C_VEL
LIN {X 0,Y 480.755,Z 815.667,A -85,B 0,C 180,E1 -6795.75,E2 -6795.75} C_VEL
LIN {X 0,Y 480.8,Z 814.777,A -85,B 0,C 180,E1 -6796.957,E2 -6796.957} C_VEL
LIN {X 0,Y 480.849,Z 813.003,A -85,B 0,C 180,E1 -6798.192,E2 -6798.192} C_VEL
LIN {X 0,Y 480.951,Z 810.269,A -85,B 0,C 180,E1 -6799.45,E2 -6799.45} C_VEL
LIN {X 0,Y 481.071,Z 806.425,A -85,B 0,C 180,E1 -6800.738,E2 -6800.738} C_VEL
LIN {X 0,Y 481.239,Z 800.807,A -85,B 0,C 180,E1 -6802.167,E2 -6802.167} C_VEL
LIN {X 0,Y 481.516,Z 793.322,A -85,B 0,C 180,E1 -6803.62,E2 -6803.62} C_VEL
LIN {X 0,Y 481.86,Z 784.907,A -85,B 0,C 180,E1 -6804.915,E2 -6804.915} C_VEL
LIN {X 0,Y 482.239,Z 776.112,A -85,B 0,C 180,E1 -6806.003,E2 -6806.003} C_VEL
LIN {X 0,Y 482.655,Z 765.872,A -85,B 0,C 180,E1 -6807.029,E2 -6807.029} C_VEL
LIN {X 0,Y 483.112,Z 754.676,A -85,B 0,C 180,E1 -6807.929,E2 -6807.929} C_VEL
LIN {X 0,Y 483.511,Z 742.593,A -85,B 0,C 180,E1 -6808.682,E2 -6808.682} C_VEL
LIN {X 0,Y 483.909,Z 729.468,A -85,B 0,C 180,E1 -6809.291,E2 -6809.291} C_VEL
LIN {X 0,Y 484.18,Z 717.5,A -85,B 0,C 180,E1 -6809.679,E2 -6809.679} C_VEL
LIN {X 0,Y 484.339,Z 702.827,A -85,B 0,C 180,E1 -6809.96,E2 -6809.96} C_VEL
LIN {X 0,Y 484.947,Z 619.175,A -85,B 0,C 180,E1 -6811.234,E2 -6811.234} C_VEL
LIN {X 0,Y 482.41,Z 606.443,A -85,B 0,C 180,E1 -6811.533,E2 -6811.533} C_VEL
LIN {X 0,Y 482.711,Z 596.977,A -85,B 0,C 180,E1 -6813.637,E2 -6813.637} C_VEL
LIN {X 0,Y 481.726,Z 590.481,A -85,B 0,C 180,E1 -6815.201,E2 -6815.201} C_VEL
LIN {X 0,Y 481.636,Z 590.493,A -85,B 0,C 180,E1 -6818.605,E2 -6818.605} C_VEL
LIN {X 0,Y 481.695,Z 590.481,A -85,B 0,C 180,E1 -6821.502,E2 -6821.502} C_VEL
LIN {X 0,Y 481.732,Z 590.482,A -85,B 0,C 180,E1 -6824.776,E2 -6824.776} C_VEL
LIN {X 0,Y 481.785,Z 590.471,A -85,B 0,C 180,E1 -6828.216,E2 -6828.216} C_VEL
LIN {X 0,Y 481.754,Z 590.473,A -85,B 0,C 180,E1 -6831.612,E2 -6831.612} C_VEL
LIN {X 0,Y 481.821,Z 590.465,A -85,B 0,C 180,E1 -6834.14,E2 -6834.14} C_VEL
LIN {X 0,Y 481.925,Z 590.452,A -85,B 0,C 180,E1 -6837.493,E2 -6837.493} C_VEL
LIN {X 0,Y 481.93,Z 590.45,A -85,B 0,C 180,E1 -6840,E2 -6840} C_VEL
LIN {X 0,Y 481.92,Z 590.454,A -85,B 0,C 180,E1 -6842.508,E2 -6842.508} C_VEL
LIN {X 0,Y 481.822,Z 590.463,A -85,B 0,C 180,E1 -6845.861,E2 -6845.861} C_VEL
LIN {X 0,Y 481.755,Z 590.473,A -85,B 0,C 180,E1 -6848.389,E2 -6848.389} C_VEL
LIN {X 0,Y 481.787,Z 590.467,A -85,B 0,C 180,E1 -6851.784,E2 -6851.784} C_VEL
LIN {X 0,Y 481.733,Z 590.478,A -85,B 0,C 180,E1 -6855.225,E2 -6855.225} C_VEL
LIN {X 0,Y 481.704,Z 590.481,A -85,B 0,C 180,E1 -6858.722,E2 -6858.722} C_VEL
LIN {X 0,Y 481.637,Z 590.489,A -85,B 0,C 180,E1 -6861.396,E2 -6861.396} C_VEL
LIN {X 0,Y 481.669,Z 590.482,A -85,B 0,C 180,E1 -6864.114,E2 -6864.114} C_VEL
LIN {X 0,Y 481.745,Z 590.477,A -85,B 0,C 180,E1 -6867.141,E2 -6867.141} C_VEL
LIN {X 0,Y 481.682,Z 590.481,A -85,B 0,C 180,E1 -6869.741,E2 -6869.741} C_VEL
LIN {X 0,Y 481.667,Z 590.48,A -85,B 0,C 180,E1 -6872.675,E2 -6872.675} C_VEL
LIN {X 0,Y 481.638,Z 590.489,A -85,B 0,C 180,E1 -6875.71,E2 -6875.71} C_VEL
LIN {X 0,Y 481.668,Z 590.482,A -85,B 0,C 180,E1 -6878.86,E2 -6878.86} C_VEL
LIN {X 0,Y 481.658,Z 590.486,A -85,B 0,C 180,E1 -6881.915,E2 -6881.915} C_VEL
LIN {X 0,Y 481.657,Z 590.484,A -85,B 0,C 180,E1 -6884.458,E2 -6884.458} C_VEL
LIN {X 0,Y 481.646,Z 590.49,A -85,B 0,C 180,E1 -6887.84,E2 -6887.84} C_VEL
LIN {X 0,Y 481.712,Z 590.477,A -85,B 0,C 180,E1 -6890.647,E2 -6890.647} C_VEL
LIN {X 0,Y 481.642,Z 590.487,A -85,B 0,C 180,E1 -6894.292,E2 -6894.292} C_VEL
LIN {X 0,Y 481.672,Z 590.489,A -85,B 0,C 180,E1 -6897.327,E2 -6897.327} C_VEL
LIN {X 0,Y 481.679,Z 590.485,A -85,B 0,C 180,E1 -6900.26,E2 -6900.26} C_VEL
LIN {X 0,Y 481.732,Z 590.482,A -85,B 0,C 180,E1 -6903.58,E2 -6903.58} C_VEL
LIN {X 0,Y 481.775,Z 590.749,A -85,B 0,C 180,E1 -6903.757,E2 -6903.757} C_VEL
LIN {X 0,Y 483.921,Z 601.909,A -85,B 0,C 180,E1 -6905.779,E2 -6905.779} C_VEL
LIN {X 0,Y 483.762,Z 611.315,A -85,B 0,C 180,E1 -6907.358,E2 -6907.358} C_VEL
LIN {X 0,Y 482.915,Z 632.555,A -85,B 0,C 180,E1 -6910.842,E2 -6910.842} C_VEL
LIN {X 0,Y 482.341,Z 649.086,A -85,B 0,C 180,E1 -6913.491,E2 -6913.491} C_VEL
LIN {X 0,Y 484.776,Z 666.696,A -85,B 0,C 180,E1 -6913.848,E2 -6913.848} C_VEL
LIN {X 0,Y 484.122,Z 758.216,A -85,B 0,C 180,E1 -6915.256,E2 -6915.256} C_VEL
LIN {X 0,Y 483.826,Z 772.056,A -85,B 0,C 180,E1 -6915.65,E2 -6915.65} C_VEL
LIN {X 0,Y 483.468,Z 784.5,A -85,B 0,C 180,E1 -6916.176,E2 -6916.176} C_VEL
LIN {X 0,Y 483.005,Z 796.429,A -85,B 0,C 180,E1 -6916.859,E2 -6916.859} C_VEL
LIN {X 0,Y 482.568,Z 807.902,A -85,B 0,C 180,E1 -6917.702,E2 -6917.702} C_VEL
LIN {X 0,Y 482.154,Z 818.259,A -85,B 0,C 180,E1 -6918.652,E2 -6918.652} C_VEL
LIN {X 0,Y 481.753,Z 827.557,A -85,B 0,C 180,E1 -6919.706,E2 -6919.706} C_VEL
LIN {X 0,Y 481.407,Z 836.61,A -85,B 0,C 180,E1 -6920.971,E2 -6920.971} C_VEL
LIN {X 0,Y 481.149,Z 843.902,A -85,B 0,C 180,E1 -6922.235,E2 -6922.235} C_VEL
LIN {X 0,Y 480.952,Z 849.923,A -85,B 0,C 180,E1 -6923.549,E2 -6923.549} C_VEL
LIN {X 0,Y 480.905,Z 854.94,A -85,B 0,C 180,E1 -6924.97,E2 -6924.97} C_VEL
LIN {X 0,Y 480.846,Z 857.267,A -85,B 0,C 180,E1 -6925.809,E2 -6925.809} C_VEL
LIN {X 0,Y 480.892,Z 859.161,A -85,B 0,C 180,E1 -6926.649,E2 -6926.649} C_VEL
LIN {X 0,Y 480.845,Z 860.575,A -85,B 0,C 180,E1 -6927.487,E2 -6927.487} C_VEL
LIN {X 0,Y 480.823,Z 861.587,A -85,B 0,C 180,E1 -6928.325,E2 -6928.325} C_VEL
LIN {X 0,Y 480.743,Z 862.431,A -85,B 0,C 180,E1 -6930,E2 -6930} C_VEL
LIN {X 0,Y 480.823,Z 861.613,A -85,B 0,C 180,E1 -6931.675,E2 -6931.675} C_VEL
LIN {X 0,Y 480.845,Z 860.614,A -85,B 0,C 180,E1 -6932.513,E2 -6932.513} C_VEL
LIN {X 0,Y 480.892,Z 859.21,A -85,B 0,C 180,E1 -6933.351,E2 -6933.351} C_VEL
LIN {X 0,Y 480.851,Z 856.249,A -85,B 0,C 180,E1 -6934.611,E2 -6934.611} C_VEL
LIN {X 0,Y 480.952,Z 852.245,A -85,B 0,C 180,E1 -6935.871,E2 -6935.871} C_VEL
LIN {X 0,Y 481.109,Z 846.079,A -85,B 0,C 180,E1 -6937.343,E2 -6937.343} C_VEL
LIN {X 0,Y 481.339,Z 839.346,A -85,B 0,C 180,E1 -6938.607,E2 -6938.607} C_VEL
LIN {X 0,Y 481.611,Z 830.99,A -85,B 0,C 180,E1 -6939.873,E2 -6939.873} C_VEL
LIN {X 0,Y 481.984,Z 822.41,A -85,B 0,C 180,E1 -6940.927,E2 -6940.927} C_VEL
LIN {X 0,Y 482.469,Z 811.831,A -85,B 0,C 180,E1 -6941.979,E2 -6941.979} C_VEL
LIN {X 0,Y 482.83,Z 800.543,A -85,B 0,C 180,E1 -6942.884,E2 -6942.884} C_VEL
LIN {X 0,Y 483.256,Z 789.805,A -85,B 0,C 180,E1 -6943.562,E2 -6943.562} C_VEL
LIN {X 0,Y 483.7,Z 776.57,A -85,B 0,C 180,E1 -6944.193,E2 -6944.193} C_VEL
LIN {X 0,Y 484.084,Z 763.184,A -85,B 0,C 180,E1 -6944.637,E2 -6944.637} C_VEL
LIN {X 0,Y 484.305,Z 748.073,A -85,B 0,C 180,E1 -6944.926,E2 -6944.926} C_VEL
LIN {X 0,Y 484.686,Z 664.831,A -85,B 0,C 180,E1 -6946.189,E2 -6946.189} C_VEL
LIN {X 0,Y 482.376,Z 649.245,A -85,B 0,C 180,E1 -6946.533,E2 -6946.533} C_VEL
LIN {X 0,Y 483.084,Z 629.331,A -85,B 0,C 180,E1 -6949.769,E2 -6949.769} C_VEL
LIN {X 0,Y 483.798,Z 611.912,A -85,B 0,C 180,E1 -6952.641,E2 -6952.641} C_VEL
LIN {X 0,Y 484.08,Z 602.525,A -85,B 0,C 180,E1 -6954.213,E2 -6954.213} C_VEL
LIN {X 0,Y 481.732,Z 590.482,A -85,B 0,C 180,E1 -6956.42,E2 -6956.42} C_VEL
LIN {X 0,Y 481.679,Z 590.484,A -85,B 0,C 180,E1 -6959.74,E2 -6959.74} C_VEL
LIN {X 0,Y 481.672,Z 590.487,A -85,B 0,C 180,E1 -6962.673,E2 -6962.673} C_VEL
LIN {X 0,Y 481.642,Z 590.485,A -85,B 0,C 180,E1 -6965.708,E2 -6965.708} C_VEL
LIN {X 0,Y 481.712,Z 590.476,A -85,B 0,C 180,E1 -6969.353,E2 -6969.353} C_VEL
LIN {X 0,Y 481.646,Z 590.487,A -85,B 0,C 180,E1 -6972.16,E2 -6972.16} C_VEL
LIN {X 0,Y 481.657,Z 590.482,A -85,B 0,C 180,E1 -6975.542,E2 -6975.542} C_VEL
LIN {X 0,Y 481.658,Z 590.484,A -85,B 0,C 180,E1 -6978.085,E2 -6978.085} C_VEL
LIN {X 0,Y 481.667,Z 590.485,A -85,B 0,C 180,E1 -6981.14,E2 -6981.14} C_VEL
LIN {X 0,Y 481.663,Z 590.491,A -85,B 0,C 180,E1 -6984.794,E2 -6984.794} C_VEL
LIN {X 0,Y 481.667,Z 590.484,A -85,B 0,C 180,E1 -6987.325,E2 -6987.325} C_VEL
LIN {X 0,Y 481.682,Z 590.48,A -85,B 0,C 180,E1 -6990.259,E2 -6990.259} C_VEL
LIN {X 0,Y 481.745,Z 590.478,A -85,B 0,C 180,E1 -6993.112,E2 -6993.112} C_VEL
LIN {X 0,Y 481.669,Z 590.481,A -85,B 0,C 180,E1 -6995.886,E2 -6995.886} C_VEL
LIN {X 0,Y 481.694,Z 590.486,A -85,B 0,C 180,E1 -6999.027,E2 -6999.027} C_VEL
LIN {X 0,Y 481.699,Z 590.477,A -85,B 0,C 180,E1 -7002.158,E2 -7002.158} C_VEL
LIN {X 0,Y 481.733,Z 590.476,A -85,B 0,C 180,E1 -7004.775,E2 -7004.775} C_VEL
LIN {X 0,Y 481.743,Z 590.471,A -85,B 0,C 180,E1 -7008.214,E2 -7008.214} C_VEL
LIN {X 0,Y 481.754,Z 590.475,A -85,B 0,C 180,E1 -7011.611,E2 -7011.611} C_VEL
LIN {X 0,Y 481.815,Z 590.463,A -85,B 0,C 180,E1 -7014.139,E2 -7014.139} C_VEL
LIN {X 0,Y 481.919,Z 590.458,A -85,B 0,C 180,E1 -7017.492,E2 -7017.492} C_VEL
LIN {X 0,Y 481.93,Z 590.45,A -85,B 0,C 180,E1 -7020,E2 -7020} C_VEL
LIN {X 0,Y 481.919,Z 590.45,A -85,B 0,C 180,E1 -7022.507,E2 -7022.507} C_VEL
LIN {X 0,Y 481.818,Z 590.467,A -85,B 0,C 180,E1 -7025.86,E2 -7025.86} C_VEL
LIN {X 0,Y 481.753,Z 590.471,A -85,B 0,C 180,E1 -7028.388,E2 -7028.388} C_VEL
LIN {X 0,Y 481.742,Z 590.479,A -85,B 0,C 180,E1 -7031.785,E2 -7031.785} C_VEL
LIN {X 0,Y 481.731,Z 590.475,A -85,B 0,C 180,E1 -7035.224,E2 -7035.224} C_VEL
LIN {X 0,Y 481.702,Z 590.477,A -85,B 0,C 180,E1 -7038.722,E2 -7038.722} C_VEL
LIN {X 0,Y 481.635,Z 590.488,A -85,B 0,C 180,E1 -7041.395,E2 -7041.395} C_VEL
LIN {X 0,Y 481.667,Z 590.487,A -85,B 0,C 180,E1 -7044.113,E2 -7044.113} C_VEL
LIN {X 0,Y 481.742,Z 590.472,A -85,B 0,C 180,E1 -7047.141,E2 -7047.141} C_VEL
LIN {X 0,Y 481.678,Z 590.485,A -85,B 0,C 180,E1 -7049.741,E2 -7049.741} C_VEL
LIN {X 0,Y 481.663,Z 590.483,A -85,B 0,C 180,E1 -7052.674,E2 -7052.674} C_VEL
LIN {X 0,Y 481.634,Z 590.489,A -85,B 0,C 180,E1 -7055.709,E2 -7055.709} C_VEL
LIN {X 0,Y 481.714,Z 590.476,A -85,B 0,C 180,E1 -7059.355,E2 -7059.355} C_VEL
LIN {X 0,Y 481.667,Z 590.489,A -85,B 0,C 180,E1 -7062.158,E2 -7062.158} C_VEL
LIN {X 0,Y 481.652,Z 590.489,A -85,B 0,C 180,E1 -7064.458,E2 -7064.458} C_VEL
LIN {X 0,Y 481.646,Z 590.486,A -85,B 0,C 180,E1 -7067.84,E2 -7067.84} C_VEL
LIN {X 0,Y 481.673,Z 590.485,A -85,B 0,C 180,E1 -7070.651,E2 -7070.651} C_VEL
LIN {X 0,Y 481.625,Z 590.486,A -85,B 0,C 180,E1 -7073.376,E2 -7073.376} C_VEL
LIN {X 0,Y 481.703,Z 590.483,A -85,B 0,C 180,E1 -7076.33,E2 -7076.33} C_VEL
LIN {X 0,Y 481.645,Z 590.484,A -85,B 0,C 180,E1 -7079.418,E2 -7079.418} C_VEL
LIN {X 0,Y 481.695,Z 590.481,A -85,B 0,C 180,E1 -7082.169,E2 -7082.169} C_VEL
LIN {X 0,Y 481.713,Z 590.479,A -85,B 0,C 180,E1 -7084.97,E2 -7084.97} C_VEL
LIN {X 0,Y 481.634,Z 590.486,A -85,B 0,C 180,E1 -7087.993,E2 -7087.993} C_VEL
LIN {X 0,Y 480.966,Z 590.578,A -85,B 0,C 180,E1 -7088.691,E2 -7088.691} C_VEL
LIN {X 0,Y 478.137,Z 590.925,A -85,B 0,C 180,E1 -7089.825,E2 -7089.825} C_VEL
LIN {X 0,Y 475.753,Z 591.227,A -85,B 0,C 180,E1 -7090.739,E2 -7090.739} C_VEL
LIN {X 0,Y 474.733,Z 591.346,A -85,B 0,C 180,E1 -7091.445,E2 -7091.445} C_VEL
LIN {X 0,Y 474.652,Z 591.355,A -85,B 0,C 180,E1 -7091.684,E2 -7091.684} C_VEL
LIN {X 0,Y 474.696,Z 591.355,A -85,B 0,C 180,E1 -7094.545,E2 -7094.545} C_VEL
LIN {X 0,Y 474.701,Z 591.349,A -85,B 0,C 180,E1 -7098.038,E2 -7098.038} C_VEL
LIN {X 0,Y 474.725,Z 591.348,A -85,B 0,C 180,E1 -7101.487,E2 -7101.487} C_VEL
LIN {X 0,Y 474.767,Z 591.341,A -85,B 0,C 180,E1 -7104.052,E2 -7104.052} C_VEL
LIN {X 0,Y 474.892,Z 591.328,A -85,B 0,C 180,E1 -7107.455,E2 -7107.455} C_VEL
LIN {X 0,Y 474.909,Z 591.323,A -85,B 0,C 180,E1 -7110,E2 -7110} C_VEL
LIN {X 0,Y 474.892,Z 591.327,A -85,B 0,C 180,E1 -7112.545,E2 -7112.545} C_VEL
LIN {X 0,Y 474.768,Z 591.341,A -85,B 0,C 180,E1 -7115.948,E2 -7115.948} C_VEL
LIN {X 0,Y 474.725,Z 591.347,A -85,B 0,C 180,E1 -7118.513,E2 -7118.513} C_VEL
LIN {X 0,Y 474.701,Z 591.35,A -85,B 0,C 180,E1 -7121.962,E2 -7121.962} C_VEL
LIN {X 0,Y 474.696,Z 591.357,A -85,B 0,C 180,E1 -7125.455,E2 -7125.455} C_VEL
LIN {X 0,Y 474.662,Z 591.357,A -85,B 0,C 180,E1 -7129.01,E2 -7129.01} C_VEL
LIN {X 0,Y 474.586,Z 591.369,A -85,B 0,C 180,E1 -7131.728,E2 -7131.728} C_VEL
LIN {X 0,Y 474.689,Z 591.406,A -85,B 0,C 180,E1 -7134.957,E2 -7134.957} C_VEL
LIN {X 0,Y 475.622,Z 597.206,A -85,B 0,C 180,E1 -7136.313,E2 -7136.313} C_VEL
LIN {X 0,Y 475.406,Z 606.352,A -85,B 0,C 180,E1 -7138.323,E2 -7138.323} C_VEL
LIN {X 0,Y 478.178,Z 620.859,A -85,B 0,C 180,E1 -7138.652,E2 -7138.652} C_VEL
LIN {X 0,Y 477.384,Z 713.209,A -85,B 0,C 180,E1 -7140.096,E2 -7140.096} C_VEL
LIN {X 0,Y 477.097,Z 726.572,A -85,B 0,C 180,E1 -7140.483,E2 -7140.483} C_VEL
LIN {X 0,Y 476.789,Z 738.593,A -85,B 0,C 180,E1 -7140.996,E2 -7140.996} C_VEL
LIN {X 0,Y 476.348,Z 749.601,A -85,B 0,C 180,E1 -7141.62,E2 -7141.62} C_VEL
LIN {X 0,Y 475.93,Z 760.418,A -85,B 0,C 180,E1 -7142.406,E2 -7142.406} C_VEL
LIN {X 0,Y 475.455,Z 771.418,A -85,B 0,C 180,E1 -7143.408,E2 -7143.408} C_VEL
LIN {X 0,Y 475.08,Z 780.735,A -85,B 0,C 180,E1 -7144.46,E2 -7144.46} C_VEL
LIN {X 0,Y 474.677,Z 789.214,A -85,B 0,C 180,E1 -7145.639,E2 -7145.639} C_VEL
LIN {X 0,Y 474.365,Z 796.385,A -85,B 0,C 180,E1 -7146.867,E2 -7146.867} C_VEL
LIN {X 0,Y 474.126,Z 802.735,A -85,B 0,C 180,E1 -7148.223,E2 -7148.223} C_VEL
LIN {X 0,Y 473.944,Z 807.819,A -85,B 0,C 180,E1 -7149.615,E2 -7149.615} C_VEL
LIN {X 0,Y 473.833,Z 811.221,A -85,B 0,C 180,E1 -7150.849,E2 -7150.849} C_VEL
LIN {X 0,Y 473.718,Z 813.749,A -85,B 0,C 180,E1 -7152.117,E2 -7152.117} C_VEL
LIN {X 0,Y 473.674,Z 815.335,A -85,B 0,C 180,E1 -7153.363,E2 -7153.363} C_VEL
LIN {X 0,Y 473.656,Z 816.063,A -85,B 0,C 180,E1 -7154.586,E2 -7154.586} C_VEL
LIN {X 0,Y 473.664,Z 816,A -85,B 0,C 180,E1 -7155.785,E2 -7155.785} C_VEL
LIN {X 0,Y 473.71,Z 815.142,A -85,B 0,C 180,E1 -7156.965,E2 -7156.965} C_VEL
LIN {X 0,Y 473.763,Z 813.545,A -85,B 0,C 180,E1 -7158.123,E2 -7158.123} C_VEL
LIN {X 0,Y 473.856,Z 811.235,A -85,B 0,C 180,E1 -7159.264,E2 -7159.264} C_VEL
LIN {X 0,Y 473.953,Z 808.001,A -85,B 0,C 180,E1 -7160.449,E2 -7160.449} C_VEL
LIN {X 0,Y 474.128,Z 803.239,A -85,B 0,C 180,E1 -7161.776,E2 -7161.776} C_VEL
LIN {X 0,Y 474.365,Z 796.999,A -85,B 0,C 180,E1 -7163.132,E2 -7163.132} C_VEL
LIN {X 0,Y 474.69,Z 788.975,A -85,B 0,C 180,E1 -7164.516,E2 -7164.516} C_VEL
LIN {X 0,Y 475.118,Z 779.531,A -85,B 0,C 180,E1 -7165.799,E2 -7165.799} C_VEL
LIN {X 0,Y 475.562,Z 769.918,A -85,B 0,C 180,E1 -7166.853,E2 -7166.853} C_VEL
LIN {X 0,Y 476.044,Z 759.239,A -85,B 0,C 180,E1 -7167.798,E2 -7167.798} C_VEL
LIN {X 0,Y 476.487,Z 747.869,A -85,B 0,C 180,E1 -7168.59,E2 -7168.59} C_VEL
LIN {X 0,Y 476.883,Z 735.456,A -85,B 0,C 180,E1 -7169.257,E2 -7169.257} C_VEL
LIN {X 0,Y 477.155,Z 723.212,A -85,B 0,C 180,E1 -7169.735,E2 -7169.735} C_VEL
LIN {X 0,Y 477.419,Z 709.44,A -85,B 0,C 180,E1 -7170.073,E2 -7170.073} C_VEL
LIN {X 0,Y 478.148,Z 619.898,A -85,B 0,C 180,E1 -7171.465,E2 -7171.465} C_VEL
LIN {X 0,Y 475.454,Z 606.744,A -85,B 0,C 180,E1 -7171.795,E2 -7171.795} C_VEL
LIN {X 0,Y 475.759,Z 598.316,A -85,B 0,C 180,E1 -7173.695,E2 -7173.695} C_VEL
LIN {X 0,Y 474.922,Z 592.582,A -85,B 0,C 180,E1 -7175.055,E2 -7175.055} C_VEL
LIN {X 0,Y 474.661,Z 591.361,A -85,B 0,C 180,E1 -7175.391,E2 -7175.391} C_VEL
LIN {X 0,Y 474.66,Z 591.358,A -85,B 0,C 180,E1 -7179.185,E2 -7179.185} C_VEL
LIN {X 0,Y 474.647,Z 591.359,A -85,B 0,C 180,E1 -7181.884,E2 -7181.884} C_VEL
LIN {X 0,Y 474.689,Z 591.36,A -85,B 0,C 180,E1 -7184.544,E2 -7184.544} C_VEL
LIN {X 0,Y 474.728,Z 591.349,A -85,B 0,C 180,E1 -7188.039,E2 -7188.039} C_VEL
LIN {X 0,Y 474.719,Z 591.35,A -85,B 0,C 180,E1 -7191.487,E2 -7191.487} C_VEL
LIN {X 0,Y 474.782,Z 591.341,A -85,B 0,C 180,E1 -7194.053,E2 -7194.053} C_VEL
LIN {X 0,Y 474.892,Z 591.328,A -85,B 0,C 180,E1 -7197.456,E2 -7197.456} C_VEL
LIN {X 0,Y 474.867,Z 591.335,A -85,B 0,C 180,E1 -7200.848,E2 -7200.848} C_VEL
LIN {X 0,Y 474.886,Z 591.33,A -85,B 0,C 180,E1 -7202.545,E2 -7202.545} C_VEL
LIN {X 0,Y 474.782,Z 591.34,A -85,B 0,C 180,E1 -7205.948,E2 -7205.948} C_VEL
LIN {X 0,Y 474.72,Z 591.35,A -85,B 0,C 180,E1 -7208.514,E2 -7208.514} C_VEL
LIN {X 0,Y 474.73,Z 591.346,A -85,B 0,C 180,E1 -7211.962,E2 -7211.962} C_VEL
LIN {X 0,Y 474.672,Z 591.352,A -85,B 0,C 180,E1 -7215.769,E2 -7215.769} C_VEL
LIN {X 0,Y 474.657,Z 591.36,A -85,B 0,C 180,E1 -7219.011,E2 -7219.011} C_VEL
LIN {X 0,Y 474.58,Z 591.365,A -85,B 0,C 180,E1 -7221.73,E2 -7221.73} C_VEL
LIN {X 0,Y 474.651,Z 591.357,A -85,B 0,C 180,E1 -7224.494,E2 -7224.494} C_VEL
LIN {X 0,Y 474.692,Z 591.356,A -85,B 0,C 180,E1 -7227.34,E2 -7227.34} C_VEL
LIN {X 0,Y 474.611,Z 591.362,A -85,B 0,C 180,E1 -7230.814,E2 -7230.814} C_VEL
LIN {X 0,Y 474.632,Z 591.358,A -85,B 0,C 180,E1 -7233.985,E2 -7233.985} C_VEL
LIN {X 0,Y 474.571,Z 591.368,A -85,B 0,C 180,E1 -7236.901,E2 -7236.901} C_VEL
LIN {X 0,Y 474.639,Z 591.362,A -85,B 0,C 180,E1 -7239.651,E2 -7239.651} C_VEL
LIN {X 0,Y 474.631,Z 591.361,A -85,B 0,C 180,E1 -7242.933,E2 -7242.933} C_VEL
LIN {X 0,Y 474.606,Z 591.366,A -85,B 0,C 180,E1 -7245.896,E2 -7245.896} C_VEL
LIN {X 0,Y 474.639,Z 591.361,A -85,B 0,C 180,E1 -7249.04,E2 -7249.04} C_VEL
LIN {X 0,Y 474.615,Z 591.367,A -85,B 0,C 180,E1 -7251.704,E2 -7251.704} C_VEL
LIN {X 0,Y 474.629,Z 591.36,A -85,B 0,C 180,E1 -7254.727,E2 -7254.727} C_VEL
LIN {X 0,Y 474.636,Z 591.365,A -85,B 0,C 180,E1 -7257.789,E2 -7257.789} C_VEL
LIN {X 0,Y 474.624,Z 591.363,A -85,B 0,C 180,E1 -7260.885,E2 -7260.885} C_VEL
LIN {X 0,Y 474.715,Z 591.507,A -85,B 0,C 180,E1 -7263.514,E2 -7263.514} C_VEL
LIN {X 0,Y 476.934,Z 602.955,A -85,B 0,C 180,E1 -7265.632,E2 -7265.632} C_VEL
LIN {X 0,Y 477.041,Z 606.566,A -85,B 0,C 180,E1 -7266.257,E2 -7266.257} C_VEL
LIN {X 0,Y 476.298,Z 623.087,A -85,B 0,C 180,E1 -7269.034,E2 -7269.034} C_VEL
LIN {X 0,Y 475.574,Z 641.872,A -85,B 0,C 180,E1 -7272.143,E2 -7272.143} C_VEL
LIN {X 0,Y 475.34,Z 648.485,A -85,B 0,C 180,E1 -7273.228,E2 -7273.228} C_VEL
LIN {X 0,Y 477.96,Z 667.373,A -85,B 0,C 180,E1 -7273.626,E2 -7273.626} C_VEL
LIN {X 0,Y 477.258,Z 757.665,A -85,B 0,C 180,E1 -7275.039,E2 -7275.039} C_VEL
LIN {X 0,Y 476.95,Z 771.552,A -85,B 0,C 180,E1 -7275.439,E2 -7275.439} C_VEL
LIN {X 0,Y 476.567,Z 784.029,A -85,B 0,C 180,E1 -7275.972,E2 -7275.972} C_VEL
LIN {X 0,Y 476.117,Z 794.699,A -85,B 0,C 180,E1 -7276.579,E2 -7276.579} C_VEL
LIN {X 0,Y 475.701,Z 805.277,A -85,B 0,C 180,E1 -7277.34,E2 -7277.34} C_VEL
LIN {X 0,Y 475.282,Z 815.684,A -85,B 0,C 180,E1 -7278.269,E2 -7278.269} C_VEL
LIN {X 0,Y 474.772,Z 825.433,A -85,B 0,C 180,E1 -7279.337,E2 -7279.337} C_VEL
LIN {X 0,Y 474.467,Z 833.434,A -85,B 0,C 180,E1 -7280.408,E2 -7280.408} C_VEL
LIN {X 0,Y 474.179,Z 841.255,A -85,B 0,C 180,E1 -7281.691,E2 -7281.691} C_VEL
LIN {X 0,Y 473.927,Z 848.45,A -85,B 0,C 180,E1 -7283.187,E2 -7283.187} C_VEL
LIN {X 0,Y 473.874,Z 853.247,A -85,B 0,C 180,E1 -7284.468,E2 -7284.468} C_VEL
LIN {X 0,Y 473.751,Z 856.91,A -85,B 0,C 180,E1 -7285.746,E2 -7285.746} C_VEL
LIN {X 0,Y 473.818,Z 858.808,A -85,B 0,C 180,E1 -7286.599,E2 -7286.599} C_VEL
LIN {X 0,Y 473.756,Z 861.242,A -85,B 0,C 180,E1 -7288.3,E2 -7288.3} C_VEL
LIN {X 0,Y 473.669,Z 862.088,A -85,B 0,C 180,E1 -7290,E2 -7290} C_VEL
LIN {X 0,Y 473.756,Z 861.272,A -85,B 0,C 180,E1 -7291.7,E2 -7291.7} C_VEL
LIN {X 0,Y 473.761,Z 860.272,A -85,B 0,C 180,E1 -7292.551,E2 -7292.551} C_VEL
LIN {X 0,Y 473.799,Z 858.866,A -85,B 0,C 180,E1 -7293.401,E2 -7293.401} C_VEL
LIN {X 0,Y 473.773,Z 855.904,A -85,B 0,C 180,E1 -7294.68,E2 -7294.68} C_VEL
LIN {X 0,Y 473.858,Z 851.895,A -85,B 0,C 180,E1 -7295.959,E2 -7295.959} C_VEL
LIN {X 0,Y 474.018,Z 845.722,A -85,B 0,C 180,E1 -7297.454,E2 -7297.454} C_VEL
LIN {X 0,Y 474.287,Z 838.984,A -85,B 0,C 180,E1 -7298.736,E2 -7298.736} C_VEL
LIN {X 0,Y 474.576,Z 830.621,A -85,B 0,C 180,E1 -7300.021,E2 -7300.021} C_VEL
LIN {X 0,Y 474.958,Z 822.028,A -85,B 0,C 180,E1 -7301.09,E2 -7301.09} C_VEL
LIN {X 0,Y 475.462,Z 811.658,A -85,B 0,C 180,E1 -7302.138,E2 -7302.138} C_VEL
LIN {X 0,Y 475.829,Z 801.213,A -85,B 0,C 180,E1 -7302.995,E2 -7302.995} C_VEL
LIN {X 0,Y 476.332,Z 789.376,A -85,B 0,C 180,E1 -7303.763,E2 -7303.763} C_VEL
LIN {X 0,Y 476.773,Z 777.41,A -85,B 0,C 180,E1 -7304.349,E2 -7304.349} C_VEL
LIN {X 0,Y 477.16,Z 764.508,A -85,B 0,C 180,E1 -7304.8,E2 -7304.8} C_VEL
LIN {X 0,Y 477.425,Z 750.925,A -85,B 0,C 180,E1 -7305.092,E2 -7305.092} C_VEL
LIN {X 0,Y 477.882,Z 665.744,A -85,B 0,C 180,E1 -7306.407,E2 -7306.407} C_VEL
LIN {X 0,Y 475.392,Z 648.958,A -85,B 0,C 180,E1 -7306.778,E2 -7306.778} C_VEL
LIN {X 0,Y 476.103,Z 630.36,A -85,B 0,C 180,E1 -7309.847,E2 -7309.847} C_VEL
LIN {X 0,Y 476.853,Z 612.961,A -85,B 0,C 180,E1 -7312.76,E2 -7312.76} C_VEL
LIN {X 0,Y 477.096,Z 603.567,A -85,B 0,C 180,E1 -7314.359,E2 -7314.359} C_VEL
LIN {X 0,Y 474.691,Z 591.358,A -85,B 0,C 180,E1 -7316.636,E2 -7316.636} C_VEL
LIN {X 0,Y 474.621,Z 591.363,A -85,B 0,C 180,E1 -7319.251,E2 -7319.251} C_VEL
LIN {X 0,Y 474.615,Z 591.369,A -85,B 0,C 180,E1 -7322.43,E2 -7322.43} C_VEL
LIN {X 0,Y 474.619,Z 591.359,A -85,B 0,C 180,E1 -7325.469,E2 -7325.469} C_VEL
LIN {X 0,Y 474.621,Z 591.367,A -85,B 0,C 180,E1 -7328.455,E2 -7328.455} C_VEL
LIN {X 0,Y 474.639,Z 591.36,A -85,B 0,C 180,E1 -7330.96,E2 -7330.96} C_VEL
LIN {X 0,Y 474.606,Z 591.363,A -85,B 0,C 180,E1 -7334.104,E2 -7334.104} C_VEL
LIN {X 0,Y 474.632,Z 591.361,A -85,B 0,C 180,E1 -7337.067,E2 -7337.067} C_VEL
LIN {X 0,Y 474.657,Z 591.359,A -85,B 0,C 180,E1 -7340.455,E2 -7340.455} C_VEL
LIN {X 0,Y 474.588,Z 591.363,A -85,B 0,C 180,E1 -7343.676,E2 -7343.676} C_VEL
LIN {X 0,Y 474.637,Z 591.365,A -85,B 0,C 180,E1 -7346.779,E2 -7346.779} C_VEL
LIN {X 0,Y 474.61,Z 591.36,A -85,B 0,C 180,E1 -7349.77,E2 -7349.77} C_VEL
LIN {X 0,Y 474.708,Z 591.353,A -85,B 0,C 180,E1 -7352.68,E2 -7352.68} C_VEL
LIN {X 0,Y 474.651,Z 591.357,A -85,B 0,C 180,E1 -7355.506,E2 -7355.506} C_VEL
LIN {X 0,Y 474.662,Z 591.361,A -85,B 0,C 180,E1 -7359.185,E2 -7359.185} C_VEL
LIN {X 0,Y 474.648,Z 591.356,A -85,B 0,C 180,E1 -7361.884,E2 -7361.884} C_VEL
LIN {X 0,Y 474.691,Z 591.351,A -85,B 0,C 180,E1 -7364.544,E2 -7364.544} C_VEL
LIN {X 0,Y 474.696,Z 591.35,A -85,B 0,C 180,E1 -7368.037,E2 -7368.037} C_VEL
LIN {X 0,Y 474.72,Z 591.353,A -85,B 0,C 180,E1 -7371.486,E2 -7371.486} C_VEL
LIN {X 0,Y 474.776,Z 591.34,A -85,B 0,C 180,E1 -7374.052,E2 -7374.052} C_VEL
LIN {X 0,Y 474.885,Z 591.334,A -85,B 0,C 180,E1 -7377.455,E2 -7377.455} C_VEL
LIN {X 0,Y 474.867,Z 591.329,A -85,B 0,C 180,E1 -7380.848,E2 -7380.848} C_VEL
LIN {X 0,Y 474.885,Z 591.326,A -85,B 0,C 180,E1 -7382.544,E2 -7382.544} C_VEL
LIN {X 0,Y 474.779,Z 591.343,A -85,B 0,C 180,E1 -7385.947,E2 -7385.947} C_VEL
LIN {X 0,Y 474.719,Z 591.347,A -85,B 0,C 180,E1 -7388.513,E2 -7388.513} C_VEL
LIN {X 0,Y 474.695,Z 591.354,A -85,B 0,C 180,E1 -7391.962,E2 -7391.962} C_VEL
LIN {X 0,Y 474.689,Z 591.355,A -85,B 0,C 180,E1 -7395.456,E2 -7395.456} C_VEL
LIN {X 0,Y 474.655,Z 591.355,A -85,B 0,C 180,E1 -7399.01,E2 -7399.01} C_VEL
LIN {X 0,Y 474.579,Z 591.371,A -85,B 0,C 180,E1 -7401.729,E2 -7401.729} C_VEL
LIN {X 0,Y 474.649,Z 591.357,A -85,B 0,C 180,E1 -7404.493,E2 -7404.493} C_VEL
LIN {X 0,Y 474.689,Z 591.352,A -85,B 0,C 180,E1 -7407.339,E2 -7407.339} C_VEL
LIN {X 0,Y 474.6,Z 591.362,A -85,B 0,C 180,E1 -7410.811,E2 -7410.811} C_VEL
LIN {X 0,Y 474.629,Z 591.366,A -85,B 0,C 180,E1 -7413.984,E2 -7413.984} C_VEL
LIN {X 0,Y 474.567,Z 591.366,A -85,B 0,C 180,E1 -7416.9,E2 -7416.9} C_VEL
LIN {X 0,Y 474.658,Z 591.356,A -85,B 0,C 180,E1 -7419.654,E2 -7419.654} C_VEL
LIN {X 0,Y 474.644,Z 591.357,A -85,B 0,C 180,E1 -7422.93,E2 -7422.93} C_VEL
LIN {X 0,Y 474.607,Z 591.364,A -85,B 0,C 180,E1 -7425.896,E2 -7425.896} C_VEL
LIN {X 0,Y 474.625,Z 591.359,A -85,B 0,C 180,E1 -7429.04,E2 -7429.04} C_VEL
LIN {X 0,Y 474.603,Z 591.362,A -85,B 0,C 180,E1 -7431.704,E2 -7431.704} C_VEL
LIN {X 0,Y 474.624,Z 591.363,A -85,B 0,C 180,E1 -7434.727,E2 -7434.727} C_VEL
LIN {X 0,Y 474.631,Z 591.358,A -85,B 0,C 180,E1 -7437.788,E2 -7437.788} C_VEL
LIN {X 0,Y 474.618,Z 591.363,A -85,B 0,C 180,E1 -7440.885,E2 -7440.885} C_VEL
LIN {X 0,Y 474.655,Z 591.354,A -85,B 0,C 180,E1 -7443.629,E2 -7443.629} C_VEL
LIN {X 0,Y 474.631,Z 591.367,A -85,B 0,C 180,E1 -7446.642,E2 -7446.642} C_VEL
LIN {X 0,Y 474.653,Z 591.356,A -85,B 0,C 180,E1 -7450.09,E2 -7450.09} C_VEL
LIN {X 0,Y 474.652,Z 591.355,A -85,B 0,C 180,E1 -7451.684,E2 -7451.684} C_VEL
LIN {X 0,Y 473.989,Z 591.443,A -85,B 0,C 180,E1 -7452.393,E2 -7452.393} C_VEL
LIN {X 0,Y 471.137,Z 591.797,A -85,B 0,C 180,E1 -7453.544,E2 -7453.544} C_VEL
LIN {X 0,Y 468.72,Z 592.099,A -85,B 0,C 180,E1 -7454.473,E2 -7454.473} C_VEL
LIN {X 0,Y 467.681,Z 592.228,A -85,B 0,C 180,E1 -7455.19,E2 -7455.19} C_VEL
LIN {X 0,Y 467.595,Z 592.235,A -85,B 0,C 180,E1 -7455.433,E2 -7455.433} C_VEL
LIN {X 0,Y 467.65,Z 592.234,A -85,B 0,C 180,E1 -7458.734,E2 -7458.734} C_VEL
LIN {X 0,Y 467.746,Z 592.216,A -85,B 0,C 180,E1 -7462.228,E2 -7462.228} C_VEL
LIN {X 0,Y 467.72,Z 592.225,A -85,B 0,C 180,E1 -7464.828,E2 -7464.828} C_VEL
LIN {X 0,Y 467.857,Z 592.205,A -85,B 0,C 180,E1 -7467.417,E2 -7467.417} C_VEL
LIN {X 0,Y 467.88,Z 592.199,A -85,B 0,C 180,E1 -7470,E2 -7470} C_VEL
LIN {X 0,Y 467.858,Z 592.203,A -85,B 0,C 180,E1 -7472.583,E2 -7472.583} C_VEL
LIN {X 0,Y 467.732,Z 592.217,A -85,B 0,C 180,E1 -7476.037,E2 -7476.037} C_VEL
LIN {X 0,Y 467.678,Z 592.225,A -85,B 0,C 180,E1 -7478.643,E2 -7478.643} C_VEL
LIN {X 0,Y 467.652,Z 592.227,A -85,B 0,C 180,E1 -7482.145,E2 -7482.145} C_VEL
LIN {X 0,Y 467.635,Z 592.233,A -85,B 0,C 180,E1 -7485.695,E2 -7485.695} C_VEL
LIN {X 0,Y 467.614,Z 592.233,A -85,B 0,C 180,E1 -7488.765,E2 -7488.765} C_VEL
LIN {X 0,Y 467.577,Z 592.244,A -85,B 0,C 180,E1 -7491.268,E2 -7491.268} C_VEL
LIN {X 0,Y 467.662,Z 592.33,A -85,B 0,C 180,E1 -7494.794,E2 -7494.794} C_VEL
LIN {X 0,Y 468.668,Z 598.48,A -85,B 0,C 180,E1 -7496.254,E2 -7496.254} C_VEL
LIN {X 0,Y 468.428,Z 606.58,A -85,B 0,C 180,E1 -7498.067,E2 -7498.067} C_VEL
LIN {X 0,Y 471.355,Z 621.353,A -85,B 0,C 180,E1 -7498.415,E2 -7498.415} C_VEL
LIN {X 0,Y 470.519,Z 713.607,A -85,B 0,C 180,E1 -7499.883,E2 -7499.883} C_VEL
LIN {X 0,Y 470.219,Z 726.885,A -85,B 0,C 180,E1 -7500.273,E2 -7500.273} C_VEL
LIN {X 0,Y 469.891,Z 739.311,A -85,B 0,C 180,E1 -7500.814,E2 -7500.814} C_VEL
LIN {X 0,Y 469.408,Z 751.207,A -85,B 0,C 180,E1 -7501.516,E2 -7501.516} C_VEL
LIN {X 0,Y 468.911,Z 762.803,A -85,B 0,C 180,E1 -7502.398,E2 -7502.398} C_VEL
LIN {X 0,Y 468.451,Z 773.11,A -85,B 0,C 180,E1 -7503.382,E2 -7503.382} C_VEL
LIN {X 0,Y 468.006,Z 782.73,A -85,B 0,C 180,E1 -7504.527,E2 -7504.527} C_VEL
